// Enable axis
FB_MC2_Compact_M_nMC_Power_fbStartDelay_TON(IN:= TRUE, PT:= T#200MS, Q=> , ET=> );
IF FB_MC2_Compact_M_nMC_Power_fbStartDelay_TON.Q THEN
	IF _stAXIS_REF.NcToPlc.AxisID > 0 THEN
		IF (bE_StopDelay AND (bE_Stop OR _stAXIS_REF.Status.Moving)) THEN
			FB_MC2_Compact_M_nMC_Power_fbMC2_Power(Axis:= _stAXIS_REF, Enable:= bEnable, Enable_Positive:= bEnable_Positive, Enable_Negative:= bEnable_Negative, Override:= FB_MC2_Compact_M_nMC_Power_lrOverride, BufferMode:= MC_Aborting); 					
		ELSE
			FB_MC2_Compact_M_nMC_Power_fbMC2_Power(Axis:= _stAXIS_REF, Enable:= FALSE, Enable_Positive:= bEnable_Positive, Enable_Negative:= bEnable_Negative, Override:= FB_MC2_Compact_M_nMC_Power_lrOverride, BufferMode:= MC_Aborting); 					
		END_IF
	ELSE
		FB_MC2_Compact_M_nMC_Power_fbMC2_Power(Axis:= _stAXIS_REF, Enable:= FALSE, Enable_Positive:= bEnable_Positive, Enable_Negative:= bEnable_Negative, Override:= FB_MC2_Compact_M_nMC_Power_lrOverride, BufferMode:= MC_Aborting); 					
		IF bEnable THEN
			M_nMC_Power:= Tc3_HBI_System.cMAPPING_ERROR;
		END_IF
		RETURN;
	END_IF	 	
ELSE
	FB_MC2_Compact_M_nMC_Power_fbMC2_Power(Axis:= _stAXIS_REF, Enable:= FALSE, Enable_Positive:= bEnable_Positive, Enable_Negative:= bEnable_Negative, Override:= FB_MC2_Compact_M_nMC_Power_lrOverride, BufferMode:= MC_Aborting); 					
END_IF


// Error handling
IF FB_MC2_Compact_M_nMC_Power_fbMC2_Power.Error THEN
	M_nError(nErrorID:= FB_MC2_Compact_M_nMC_Power_fbMC2_Power.ErrorID);
	_sMessage:= 'Axis Power Error';
END_IF

// Local error
IF NOT _bError AND NOT _bReset THEN
	FB_MC2_Compact_M_nMC_Power_bError:= FALSE;
END_IF
IF _bError THEN
	FB_MC2_Compact_M_nMC_Power_bError:= TRUE;
END_IF

//**************************************
// Status
//**************************************
THIS^._bReady:= bEnable AND _stAXIS_REF.Status.ControlLoopClosed AND NOT FB_MC2_Compact_M_nMC_Power_bError AND FB_MC2_Compact_M_nMC_Power_fbMC2_Power.Status;	// Axis ready to run

//**************************************
// Local reset
//**************************************
FB_MC2_Compact_M_nMC_Power_arr_fb_R_TRIG[1](CLK:= bEnable);
FB_MC2_Compact_M_nMC_Power_arr_fb_R_TRIG[2](CLK:= NOT bEnable);
FB_MC2_Compact_M_nMC_Power_arr_fb_R_TRIG[3](CLK:= bE_Stop);
FB_MC2_Compact_M_nMC_Power_arr_fb_R_TRIG[4](CLK:= NOT bE_Stop);
FB_MC2_Compact_M_nMC_Power_arr_fb_R_TRIG[5](CLK:= bE_StopDelay);
FB_MC2_Compact_M_nMC_Power_arr_fb_R_TRIG[6](CLK:= NOT bE_StopDelay);
FB_MC2_Compact_M_nMC_Power_arr_fb_R_TRIG[7](CLK:= NOT bEnable_Positive);
FB_MC2_Compact_M_nMC_Power_arr_fb_R_TRIG[8](CLK:= NOT bEnable_Negative);
FB_MC2_Compact_M_nMC_Power_arr_fb_R_TRIG[9](CLK:= _bAuto);
FB_MC2_Compact_M_nMC_Power_arr_fb_R_TRIG[10](CLK:= NOT _bAuto);
FB_MC2_Compact_M_nMC_Power_arr_fb_R_TRIG[11](CLK:= _bManual);
FB_MC2_Compact_M_nMC_Power_arr_fb_R_TRIG[12](CLK:= NOT _bManual);

FB_MC2_Compact_M_nMC_Power_bLocal_Halt:= FALSE;
FOR _iIdx:= 1 TO 12 DO
	IF FB_MC2_Compact_M_nMC_Power_arr_fb_R_TRIG[_iIdx].Q THEN
		FB_MC2_Compact_M_nMC_Power_bLocal_Halt:= TRUE;
	END_IF
END_FOR

//************************************
// Call methods
//************************************
IF THIS^._stAXIS_REF.Status.ControlLoopClosed THEN
 	FB_MC2_Compact_M_nMC_Power_arr_nRet[1]:= M_nMC_Local_Halt(bExecute:= NOT FB_MC2_Compact_M_nMC_QuickStop_bQuickStopRunning AND FB_MC2_Compact_M_nMC_Power_bLocal_Halt);
ELSE
	M_nMC_Local_Halt(bExecute:= FALSE);
END_IF
FB_MC2_Compact_M_nMC_Power_arr_nRet[2]:= M_nMC_ReadDriveAddress(bExecute:= bEnable);


// Error handling
IF _stAXIS_REF.Status.Error THEN
	M_nError(_stAXIS_REF.Status.ErrorID);
	M_nMC_Power:= _nErrorID;
ELSE
	FOR _iIdx:= 1 TO UINT_TO_INT(SIZEOF(FB_MC2_Compact_M_nMC_Power_arr_nRet) / SIZEOF(FB_MC2_Compact_M_nMC_Power_arr_nRet[1])) DO
		IF FB_MC2_Compact_M_nMC_Power_arr_nRet[_iIdx] > 10 THEN
			M_nError(nErrorID:= FB_MC2_Compact_M_nMC_Power_arr_nRet[_iIdx]);
			EXIT;
		END_IF
	END_FOR

	// Method return value
	IF _bError THEN
		M_nMC_Power:= _nErrorID;
	ELSE
		IF FB_MC2_Compact_M_nMC_Power_fbMC2_Power.Status THEN
			M_nMC_Power:= Tc3_HBI_System.cCOMPLETE;
		ELSE
			M_nMC_Power:= Tc3_HBI_System.cIDLE;
		END_IF
	END_IF

END_IF
END_METHOD

//	The result of the method is an unsigned double integer
//	0 = idle 
//	1 = coupled
//	2 = starting
//	3 = running
//	4 = aborted
// 	5 = no hardware connected
// 	6 = Spare
//	7 = pointer or index error
//	8 = mapping error
//	9 = parameter error
//	10 = complete
//	Any other number = ErrorID
METHOD PUBLIC M_nMC_QuickStop : UDINT
VAR_INPUT
	bExecute: BOOL;
	lrDeceleration: LREAL;
	lrJerk: LREAL;
END_VAR
// Local variable
FB_MC2_Compact_M_nMC_QuickStop_bExecute:= bExecute;
FB_MC2_Compact_M_nMC_QuickStop_lrDeceleration:= lrDeceleration;
FB_MC2_Compact_M_nMC_QuickStop_lrJerk:= lrJerk;

//**********************************
// Reset 
//**********************************
IF _bReset THEN
	IF _bError THEN
		FB_MC2_Compact_M_nMC_QuickStop_fbMC2_Stop(Axis:= _stAXIS_REF, Execute:= FALSE); 
		FB_MC2_Compact_M_nMC_QuickStop_iState:= 000;
		_sMessage:= '';
	END_IF
END_IF

//**********************************
// Wait for execute
//**********************************
IF _stAXIS_REF.NcToPlc.AxisID > 0 THEN
	FB_MC2_Compact_M_nMC_QuickStop_fbExecute_R_TRIG(CLK:= FB_MC2_Compact_M_nMC_QuickStop_bExecute);
	IF FB_MC2_Compact_M_nMC_QuickStop_fbExecute_R_TRIG.Q THEN
		FB_MC2_Compact_M_nMC_QuickStop_fbMC2_Stop(Axis:= _stAXIS_REF, Execute:= FALSE, Deceleration:= FB_MC2_Compact_M_nMC_QuickStop_lrDeceleration, Jerk:= FB_MC2_Compact_M_nMC_QuickStop_lrJerk); 
		FB_MC2_Compact_M_nMC_QuickStop_bQuickStopRunning:= TRUE;
		
		// Axis not coupled	
		IF NOT _stAXIS_REF.Status.Coupled THEN
			IF _stAXIS_REF.Status.ControlLoopClosed THEN
				IF _stAXIS_REF.Status.HasJob THEN
					FB_MC2_Compact_M_nMC_QuickStop_fbMC2_Stop.Execute:= TRUE;
					FB_MC2_Compact_M_nMC_QuickStop_iState:= 001;
				ELSE
					FB_MC2_Compact_M_nMC_QuickStop_iState:= 020;
				END_IF
			ELSE
				FB_MC2_Compact_M_nMC_QuickStop_iState:= 020;
			END_IF
		ELSE
			FB_MC2_Compact_M_nMC_QuickStop_iState:= 010;
		END_IF
	END_IF
ELSE
	FB_MC2_Compact_M_nMC_QuickStop_fbExecute_R_TRIG(CLK:= FALSE);
	FB_MC2_Compact_M_nMC_QuickStop_iState:= 000;
	IF FB_MC2_Compact_M_nMC_QuickStop_bExecute THEN
		M_nMC_QuickStop:= Tc3_HBI_System.cMAPPING_ERROR;
	END_IF
	RETURN;
END_IF


//**********************************
// Main sequence
//**********************************
CASE FB_MC2_Compact_M_nMC_QuickStop_iState OF

	000: 	// Do nothing
			FB_MC2_Compact_M_nMC_QuickStop_bQuickStopRunning:= FALSE;
	
	001:	// Stop Axis
			M_nMC_QuickStop:= Tc3_HBI_System.cRUNNING;
			FB_MC2_Compact_M_nMC_QuickStop_fbMC2_Stop(Axis:= _stAXIS_REF); 
			
			// Stop Axis
			IF _stAXIS_REF.Status.PTPmode AND _stAXIS_REF.Status.Operational THEN
				FB_MC2_Compact_M_nMC_QuickStop_fbMC2_Stop.Execute:= TRUE; 
		
				// Command aborted
				IF FB_MC2_Compact_M_nMC_QuickStop_fbMC2_Stop.CommandAborted THEN
					FB_MC2_Compact_M_nMC_QuickStop_iState:= 020;
				ELSE
					// Error handling
					IF FB_MC2_Compact_M_nMC_QuickStop_fbMC2_Stop.Error THEN
						M_nError(nErrorID:= FB_MC2_Compact_M_nMC_QuickStop_fbMC2_Stop.ErrorID);
						M_nMC_QuickStop:= FB_MC2_Compact_M_nMC_QuickStop_fbMC2_Stop.ErrorID;
						_sMessage:= 'Axis Quick Stop Error';
					ELSE
						// Done
						IF FB_MC2_Compact_M_nMC_QuickStop_fbMC2_Stop.Done THEN
							FB_MC2_Compact_M_nMC_QuickStop_fbMC2_Stop(Axis:= _stAXIS_REF, Execute:= FALSE); 
							FB_MC2_Compact_M_nMC_QuickStop_iState:= 020;
						END_IF
					END_IF
				END_IF
			ELSE
				FB_MC2_Compact_M_nMC_QuickStop_iState:= 020;
			END_IF
	
	010:	// Coupled
			M_nMC_QuickStop:= Tc3_HBI_System.cCOUPLED;
			FB_MC2_Compact_M_nMC_QuickStop_fbMC2_Stop(Axis:= _stAXIS_REF); 
			FB_MC2_Compact_M_nMC_QuickStop_bQuickStopRunning:= FALSE;

			IF NOT FB_MC2_Compact_M_nMC_QuickStop_bExecute THEN
				FB_MC2_Compact_M_nMC_QuickStop_fbMC2_Stop(Axis:= _stAXIS_REF, Execute:= FALSE); 
				FB_MC2_Compact_M_nMC_QuickStop_iState:= 000;
			END_IF	

	020:	// Done
			M_nMC_QuickStop:= Tc3_HBI_System.cCOMPLETE;
			FB_MC2_Compact_M_nMC_QuickStop_fbMC2_Stop(Axis:= _stAXIS_REF); 
			FB_MC2_Compact_M_nMC_QuickStop_bQuickStopRunning:= FALSE;

			IF FB_MC2_Compact_M_nMC_QuickStop_bExecute THEN
				IF FB_MC2_Compact_M_nMC_QuickStop_fbMC2_Stop.CommandAborted THEN
					M_nMC_QuickStop:= Tc3_HBI_System.cABORTED;
				END_IF
			ELSE
				FB_MC2_Compact_M_nMC_QuickStop_fbMC2_Stop(Axis:= _stAXIS_REF, Execute:= FALSE); 
				FB_MC2_Compact_M_nMC_QuickStop_iState:= 000;
			END_IF	
		
ELSE
	FB_MC2_Compact_M_nMC_QuickStop_iState:= 000;
END_CASE
END_METHOD

//	The result of the method is an unsigned double integer
//	0 = idle 
//	1 = coupled
//	2 = starting
//	3 = running
//	4 = aborted
// 	5 = no hardware connected
// 	6 = Spare
//	7 = pointer or index error
//	8 = mapping error
//	9 = parameter error
//	10 = complete
//	Any other number = ErrorID
METHOD PRIVATE M_nMC_ReadDriveAddress : UDINT
VAR_INPUT
	bExecute: BOOL;
END_VAR
// Local variable
FB_MC2_Compact_M_nMC_ReadDriveAddress_bExecute:= bExecute;

//**********************************
// Reset 
//**********************************
IF _bReset THEN
	FB_MC2_Compact_M_nMC_ReadDriveAddress_iState:= 000;
	_sMessage:= '';
END_IF

// Check for Axis
IF _stAXIS_REF.NcToPlc.AxisID = 0 THEN
	Tc2_System.MEMSET(destAddr:= ADR(_stDriveAddress), fillByte:= 16#00, n:= SIZEOF(_stDriveAddress));	
	FB_MC2_Compact_M_nMC_ReadDriveAddress_iState:= 000;
	IF FB_MC2_Compact_M_nMC_ReadDriveAddress_bExecute THEN
		M_nMC_ReadDriveAddress:= Tc3_HBI_System.cMAPPING_ERROR;
	END_IF
	RETURN;
END_IF

//**********************************
// Main sequence
//**********************************
CASE FB_MC2_Compact_M_nMC_ReadDriveAddress_iState OF

	000: 	// Init
			M_nMC_ReadDriveAddress:= Tc3_HBI_System.cSTARTING;
			FB_MC2_Compact_M_nMC_ReadDriveAddress_fbReadDriveAddress(Axis:= _stAXIS_REF, Execute:= FALSE);
			
			// WcState ok 
			IF NOT BIT_TO_BOOL(_stAXIS_REF.NcToPlc.StateDWord.30) AND NOT _stAXIS_REF.Status.OpMode.SimulationAxis THEN
				// Axis connected to Hardware
				IF _stAXIS_REF.NcToPlc.AxisID > 0 THEN
					FB_MC2_Compact_M_nMC_ReadDriveAddress_iState:= FB_MC2_Compact_M_nMC_ReadDriveAddress_iState +1;
				END_IF	
			END_IF	
		
	001:	// Read drive address		
			M_nMC_ReadDriveAddress:= Tc3_HBI_System.cSTARTING;
			FB_MC2_Compact_M_nMC_ReadDriveAddress_fbReadDriveAddress(Axis:= _stAXIS_REF, Execute:= TRUE);
			FB_MC2_Compact_M_nMC_ReadDriveAddress_iState:= FB_MC2_Compact_M_nMC_ReadDriveAddress_iState +1;

	002:	// Read drive address done	
			M_nMC_ReadDriveAddress:= Tc3_HBI_System.cRUNNING;
			FB_MC2_Compact_M_nMC_ReadDriveAddress_fbReadDriveAddress(Axis:= _stAXIS_REF, Execute:= TRUE);
			
			// Error
			IF FB_MC2_Compact_M_nMC_ReadDriveAddress_fbReadDriveAddress.Error THEN
				M_nError(nErrorID:= FB_MC2_Compact_M_nMC_ReadDriveAddress_fbReadDriveAddress.ErrorID);
				M_nMC_ReadDriveAddress:= FB_MC2_Compact_M_nMC_ReadDriveAddress_fbReadDriveAddress.ErrorID;
				_sMessage:= 'Axis Read Drive Address Error';
			ELSE
				// Done
				IF NOT FB_MC2_Compact_M_nMC_ReadDriveAddress_fbReadDriveAddress.Busy AND FB_MC2_Compact_M_nMC_ReadDriveAddress_fbReadDriveAddress.Done THEN
					_stDriveAddress:= FB_MC2_Compact_M_nMC_ReadDriveAddress_fbReadDriveAddress.DriveAddress;
					FB_MC2_Compact_M_nMC_ReadDriveAddress_fbReadDriveAddress(Axis:= _stAXIS_REF, Execute:= FALSE);
					FB_MC2_Compact_M_nMC_ReadDriveAddress_iState:= FB_MC2_Compact_M_nMC_ReadDriveAddress_iState +1;
				END_IF
			END_IF
	
	003: // Done
			M_nMC_ReadDriveAddress:= Tc3_HBI_System.cCOMPLETE;

ELSE
	FB_MC2_Compact_M_nMC_ReadDriveAddress_iState:= 000;
END_CASE
END_METHOD

//	The result of the method is an unsigned double integer
//	0 = idle 
//	1 = coupled
//	2 = starting
//	3 = running
//	4 = aborted
// 	5 = no hardware connected
// 	6 = Spare
//	7 = pointer or index error
//	8 = mapping error
//	9 = parameter error
//	10 = complete
//	Any other number = ErrorID
METHOD PUBLIC M_nMC_Stop : UDINT
VAR_INPUT
	bExecute: BOOL;
END_VAR
// Local variable
FB_MC2_Compact_M_nMC_Stop_bExecute:= bExecute;

//**********************************
// Reset 
//**********************************
IF _bReset THEN
	IF _bError THEN
		FB_MC2_Compact_M_nMC_Stop_fbMC2_Stop1(Axis:= _stAXIS_REF, Execute:= FALSE);
		FB_MC2_Compact_M_nMC_Stop_fbMC2_Stop2(Axis:= _stAXIS_REF, Execute:= FALSE);
		FB_MC2_Compact_M_nMC_Stop_iState:= 000;
		_sMessage:= '';
	END_IF
END_IF

//**********************************
// Wait for execute
//**********************************
IF _stAXIS_REF.NcToPlc.AxisID > 0 THEN
	FB_MC2_Compact_M_nMC_Stop_fbExecute_R_TRIG(CLK:= FB_MC2_Compact_M_nMC_Stop_bExecute);
	IF FB_MC2_Compact_M_nMC_Stop_fbExecute_R_TRIG.Q THEN
		FB_MC2_Compact_M_nMC_Stop_fbMC2_Stop1(Axis:= _stAXIS_REF, Deceleration:= _stDynamic.lrDeceleration, Jerk:= _stDynamic.lrJerk); 
		FB_MC2_Compact_M_nMC_Stop_fbMC2_Stop2(Axis:= _stAXIS_REF, Deceleration:= _stDynamic.lrDeceleration, Jerk:= _stDynamic.lrJerk); 
		
		// Axis not coupled	
		IF NOT _stAXIS_REF.Status.Coupled THEN
			IF FB_MC2_Compact_M_nMC_Stop_fbMC2_Stop1.Execute OR FB_MC2_Compact_M_nMC_Stop_fbMC2_Stop1.Busy THEN
				FB_MC2_Compact_M_nMC_Stop_fbMC2_Stop1(Axis:= _stAXIS_REF, Execute:= FALSE); 
				FB_MC2_Compact_M_nMC_Stop_fbMC2_Stop2(Axis:= _stAXIS_REF, Execute:= FALSE); 
				FB_MC2_Compact_M_nMC_Stop_fbMC2_Stop2.Execute:= TRUE;
				FB_MC2_Compact_M_nMC_Stop_iState:= 010;
			ELSE
				FB_MC2_Compact_M_nMC_Stop_fbMC2_Stop1(Axis:= _stAXIS_REF, Execute:= FALSE); 
				FB_MC2_Compact_M_nMC_Stop_fbMC2_Stop2(Axis:= _stAXIS_REF, Execute:= FALSE); 
				FB_MC2_Compact_M_nMC_Stop_fbMC2_Stop1.Execute:= TRUE;
				FB_MC2_Compact_M_nMC_Stop_iState:= 001;
			END_IF
		ELSE
			FB_MC2_Compact_M_nMC_Stop_fbMC2_Stop1(Axis:= _stAXIS_REF, Execute:= FALSE); 
			FB_MC2_Compact_M_nMC_Stop_fbMC2_Stop2(Axis:= _stAXIS_REF, Execute:= FALSE); 
			FB_MC2_Compact_M_nMC_Stop_iState:= 030;
		END_IF
	
	END_IF
ELSE
	FB_MC2_Compact_M_nMC_Stop_fbExecute_R_TRIG(CLK:= FALSE);
	FB_MC2_Compact_M_nMC_Stop_iState:= 000;
	IF FB_MC2_Compact_M_nMC_Stop_bExecute THEN
		M_nMC_Stop:= Tc3_HBI_System.cMAPPING_ERROR;
	END_IF
	RETURN;
END_IF


//**********************************
// Main sequence
//**********************************
CASE FB_MC2_Compact_M_nMC_Stop_iState OF

	000: 	// Do nothing
	
	001:	// Stop Axis1
			M_nMC_Stop:= Tc3_HBI_System.cSTARTING;
			FB_MC2_Compact_M_nMC_Stop_fbMC2_Stop1(Axis:= _stAXIS_REF);
			FB_MC2_Compact_M_nMC_Stop_fbMC2_Stop2(Axis:= _stAXIS_REF);
	
			// Command aborted
			IF FB_MC2_Compact_M_nMC_Stop_fbMC2_Stop1.CommandAborted THEN
				FB_MC2_Compact_M_nMC_Stop_fbMC2_Stop2.Execute:= FALSE;
				FB_MC2_Compact_M_nMC_Stop_iState:= 040;
			ELSE
				// Error handling
				IF FB_MC2_Compact_M_nMC_Stop_fbMC2_Stop1.Error THEN
					M_nError(FB_MC2_Compact_M_nMC_Stop_fbMC2_Stop1.ErrorID);
					M_nMC_Stop:= FB_MC2_Compact_M_nMC_Stop_fbMC2_Stop1.ErrorID;
					_sMessage:= 'Axis Stop Error';
				ELSE
					// Active
					IF FB_MC2_Compact_M_nMC_Stop_fbMC2_Stop1.Active THEN
						FB_MC2_Compact_M_nMC_Stop_iState:= 02;
					ELSE
						// Done
						IF FB_MC2_Compact_M_nMC_Stop_fbMC2_Stop1.Done THEN
							FB_MC2_Compact_M_nMC_Stop_iState:= 040;
						END_IF
					END_IF	
				END_IF
			END_IF

	002:	// Stop Axis
			M_nMC_Stop:= Tc3_HBI_System.cRUNNING;
			FB_MC2_Compact_M_nMC_Stop_fbMC2_Stop1(Axis:= _stAXIS_REF);
			FB_MC2_Compact_M_nMC_Stop_fbMC2_Stop2(Axis:= _stAXIS_REF);
	
			// Command aborted
			IF FB_MC2_Compact_M_nMC_Stop_fbMC2_Stop1.CommandAborted THEN
				FB_MC2_Compact_M_nMC_Stop_fbMC2_Stop2.Execute:= FALSE;
				FB_MC2_Compact_M_nMC_Stop_iState:= 040;
			ELSE
				// Error handling
				IF FB_MC2_Compact_M_nMC_Stop_fbMC2_Stop1.Error THEN
					M_nError(FB_MC2_Compact_M_nMC_Stop_fbMC2_Stop1.ErrorID);
					M_nMC_Stop:= FB_MC2_Compact_M_nMC_Stop_fbMC2_Stop1.ErrorID;
					_sMessage:= 'Axis Stop Error';
				ELSE
					// Done
					IF FB_MC2_Compact_M_nMC_Stop_fbMC2_Stop1.Done THEN
						FB_MC2_Compact_M_nMC_Stop_iState:= 040;
					END_IF
				END_IF
			END_IF 

	010:	// Stop Axis1
			M_nMC_Stop:= Tc3_HBI_System.cSTARTING;
			FB_MC2_Compact_M_nMC_Stop_fbMC2_Stop1(Axis:= _stAXIS_REF);
			FB_MC2_Compact_M_nMC_Stop_fbMC2_Stop2(Axis:= _stAXIS_REF);
			
			// Command aborted
			IF FB_MC2_Compact_M_nMC_Stop_fbMC2_Stop2.CommandAborted THEN
				FB_MC2_Compact_M_nMC_Stop_fbMC2_Stop1.Execute:= FALSE;
				FB_MC2_Compact_M_nMC_Stop_iState:= 040;
			ELSE
				// Error handling
				IF FB_MC2_Compact_M_nMC_Stop_fbMC2_Stop2.Error THEN
					M_nError(FB_MC2_Compact_M_nMC_Stop_fbMC2_Stop2.ErrorID);
					M_nMC_Stop:= FB_MC2_Compact_M_nMC_Stop_fbMC2_Stop2.ErrorID;
					_sMessage:= 'Axis Stop Error';
				ELSE
					// Active
					IF FB_MC2_Compact_M_nMC_Stop_fbMC2_Stop2.Active THEN
						FB_MC2_Compact_M_nMC_Stop_iState:= 011;
					ELSE
						// Done
						IF FB_MC2_Compact_M_nMC_Stop_fbMC2_Stop2.Done THEN
							FB_MC2_Compact_M_nMC_Stop_iState:= 040;
						END_IF
					END_IF	
				END_IF
			END_IF 
			
	011:	// Stop Axis2
			M_nMC_Stop:= Tc3_HBI_System.cRUNNING;
			FB_MC2_Compact_M_nMC_Stop_fbMC2_Stop1(Axis:= _stAXIS_REF);
			FB_MC2_Compact_M_nMC_Stop_fbMC2_Stop2(Axis:= _stAXIS_REF);
			
			// Command aborted
			IF FB_MC2_Compact_M_nMC_Stop_fbMC2_Stop2.CommandAborted THEN
				FB_MC2_Compact_M_nMC_Stop_fbMC2_Stop1.Execute:= FALSE;
				FB_MC2_Compact_M_nMC_Stop_iState:= 040;
			ELSE
				// Error handling
				IF FB_MC2_Compact_M_nMC_Stop_fbMC2_Stop2.Error THEN
					M_nError(FB_MC2_Compact_M_nMC_Stop_fbMC2_Stop2.ErrorID);
					M_nMC_Stop:= FB_MC2_Compact_M_nMC_Stop_fbMC2_Stop2.ErrorID;
					_sMessage:= 'Axis Stop Error';
				ELSE
					// Done
					IF FB_MC2_Compact_M_nMC_Stop_fbMC2_Stop2.Done THEN
						FB_MC2_Compact_M_nMC_Stop_iState:= 040;
					END_IF
				END_IF
			END_IF
		
	030:	// Coupled
			M_nMC_Stop:= Tc3_HBI_System.cCOUPLED;
			FB_MC2_Compact_M_nMC_Stop_fbMC2_Stop1(Axis:= _stAXIS_REF);
			FB_MC2_Compact_M_nMC_Stop_fbMC2_Stop2(Axis:= _stAXIS_REF);

			IF NOT FB_MC2_Compact_M_nMC_Stop_bExecute THEN
				FB_MC2_Compact_M_nMC_Stop_fbMC2_Stop1(Axis:= _stAXIS_REF, Execute:= FALSE);
				FB_MC2_Compact_M_nMC_Stop_fbMC2_Stop2(Axis:= _stAXIS_REF, Execute:= FALSE);
				FB_MC2_Compact_M_nMC_Stop_iState:= 000;
			END_IF	

	040:	// Done
			M_nMC_Stop:= Tc3_HBI_System.cCOMPLETE;
			FB_MC2_Compact_M_nMC_Stop_fbMC2_Stop1(Axis:= _stAXIS_REF);
			FB_MC2_Compact_M_nMC_Stop_fbMC2_Stop2(Axis:= _stAXIS_REF);

			IF FB_MC2_Compact_M_nMC_Stop_bExecute THEN
				IF FB_MC2_Compact_M_nMC_Stop_fbMC2_Stop1.Execute AND FB_MC2_Compact_M_nMC_Stop_fbMC2_Stop1.CommandAborted THEN
					M_nMC_Stop:= Tc3_HBI_System.cABORTED;
				END_IF
				IF FB_MC2_Compact_M_nMC_Stop_fbMC2_Stop2.Execute AND FB_MC2_Compact_M_nMC_Stop_fbMC2_Stop2.CommandAborted THEN
					M_nMC_Stop:= Tc3_HBI_System.cABORTED;
				END_IF
			ELSE	
				FB_MC2_Compact_M_nMC_Stop_fbMC2_Stop1(Axis:= _stAXIS_REF, Execute:= FALSE);
				FB_MC2_Compact_M_nMC_Stop_fbMC2_Stop2(Axis:= _stAXIS_REF, Execute:= FALSE);
				FB_MC2_Compact_M_nMC_Stop_iState:= 000;
			END_IF	
		
ELSE
	FB_MC2_Compact_M_nMC_Stop_iState:= 000;
END_CASE
END_METHOD

//	The result of the method is an unsigned double integer
//	0 = idle 
//	1 = coupled
//	2 = starting
//	3 = running
//	4 = aborted
// 	5 = no hardware connected
// 	6 = Spare
//	7 = pointer or index error
//	8 = mapping error
//	9 = parameter error
//	10 = complete
//	Any other number = ErrorID
METHOD PUBLIC M_nReset : UDINT
VAR_INPUT
	bExecute: BOOL;
END_VAR
// Local variable
FB_MC2_Compact_M_nReset_bExecute:= bExecute;

//**********************************
// Wait for execute
//**********************************
FB_MC2_Compact_M_nReset_fbExecute_R_TRIG(CLK:= FB_MC2_Compact_M_nReset_bExecute);
IF FB_MC2_Compact_M_nReset_fbExecute_R_TRIG.Q THEN
	FB_MC2_Compact_M_nReset_fbMC2_Reset(Axis:= _stAXIS_REF, Execute:= FALSE);
	SUPER^.M_nReset(bExecute:= FALSE);
	FB_MC2_Compact_M_nReset_iState:= 001;
	_sMessage:= '';
END_IF	


//**********************************
// Main sequence
//**********************************
CASE FB_MC2_Compact_M_nReset_iState OF

	000: 	// Do nothing
		
	001:	// Reset NC
			M_nReset:= Tc3_HBI_System.cSTARTING;
			FB_MC2_Compact_M_nReset_fbMC2_Reset(Axis:= _stAXIS_REF, Execute:= FALSE);
			
			// Check for not encoder axis
			IF _stAXIS_REF.Status.ErrorID = _stAXIS_REF.NcToPlc.ErrorCode THEN
				IF _stAXIS_REF.Status.Error THEN
					IF _stAXIS_REF.Status.Coupled THEN
						FB_MC2_Compact_M_nReset_iState:= FB_MC2_Compact_M_nReset_iState +2;
					ELSE
						IF _stAXIS_REF.Status.Error OR NOT _stAXIS_REF.Status.HasJob THEN 
							FB_MC2_Compact_M_nReset_iState:= FB_MC2_Compact_M_nReset_iState +1;
						ELSE
							FB_MC2_Compact_M_nReset_iState:= FB_MC2_Compact_M_nReset_iState +2;
						END_IF	
					END_IF
				ELSE
					FB_MC2_Compact_M_nReset_iState:= FB_MC2_Compact_M_nReset_iState +2;
				END_IF
			ELSE
				// Encoder axis
				FB_MC2_Compact_M_nReset_iState:= FB_MC2_Compact_M_nReset_iState +1;
			END_IF
	
	002:	// Reset NC
			M_nReset:= Tc3_HBI_System.cRUNNING;
			FB_MC2_Compact_M_nReset_fbMC2_Reset(Axis:= _stAXIS_REF, Execute:= TRUE); 
	
			// Error handling
			IF FB_MC2_Compact_M_nReset_fbMC2_Reset.Error THEN
				M_nError(FB_MC2_Compact_M_nReset_fbMC2_Reset.ErrorID);
				M_nReset:= FB_MC2_Compact_M_nReset_fbMC2_Reset.ErrorID;
				FB_MC2_Compact_M_nReset_iState:= FB_MC2_Compact_M_nReset_iState +1;
				_sMessage:= 'Axis Reset Error';
			ELSE
				// Done
				IF FB_MC2_Compact_M_nReset_fbMC2_Reset.Done THEN
					FB_MC2_Compact_M_nReset_iState:= FB_MC2_Compact_M_nReset_iState +1;
				END_IF
			END_IF
		
	003:	// Reset father	
			M_nReset:= Tc3_HBI_System.cRUNNING;
			FB_MC2_Compact_M_nReset_nStatus:= SUPER^.M_nReset(bExecute:= TRUE);
			
			// Error handling
			IF FB_MC2_Compact_M_nReset_nStatus > Tc3_HBI_System.cCOMPLETE THEN
				SUPER^.M_nReset(bExecute:= FALSE);		
				IF _stAXIS_REF.Status.Coupled THEN
					FB_MC2_Compact_M_nReset_iState:= 020;
				ELSE
					FB_MC2_Compact_M_nReset_iState:= 030;
				END_IF
			END_IF

			// Done
			IF FB_MC2_Compact_M_nReset_nStatus = Tc3_HBI_System.cCOUPLED OR FB_MC2_Compact_M_nReset_nStatus = Tc3_HBI_System.cCOMPLETE THEN
				SUPER^.M_nReset(bExecute:= FALSE);		
				IF _stAXIS_REF.Status.Coupled THEN
					FB_MC2_Compact_M_nReset_iState:= 020;
				ELSE
					FB_MC2_Compact_M_nReset_iState:= 030;
				END_IF
			END_IF
			
	020:	// Coupled
			M_nReset:= Tc3_HBI_System.cCOUPLED;
			IF NOT FB_MC2_Compact_M_nReset_bExecute THEN
				FB_MC2_Compact_M_nReset_fbMC2_Reset(Axis:= _stAXIS_REF, Execute:= FALSE);
				SUPER^.M_nReset(bExecute:= FALSE);		
				FB_MC2_Compact_M_nReset_iState:= 000;
			END_IF	
	
	030:	// Done
			M_nReset:= Tc3_HBI_System.cCOMPLETE;
			IF NOT FB_MC2_Compact_M_nReset_bExecute THEN
				FB_MC2_Compact_M_nReset_fbMC2_Reset(Axis:= _stAXIS_REF, Execute:= FALSE);
				SUPER^.M_nReset(bExecute:= FALSE);		
				FB_MC2_Compact_M_nReset_iState:= 000;
			END_IF

ELSE
	FB_MC2_Compact_M_nReset_iState:= 000;
END_CASE
END_METHOD

PROPERTY PUBLIC P_bE_Stop : BOOL
GET
P_bE_Stop:= FB_MC2_Compact_M_nMC_Power_bE_Stop;
END_GET
END_PROPERTY

PROPERTY PUBLIC P_bE_StopDelay : BOOL
GET
P_bE_StopDelay:= FB_MC2_Compact_M_nMC_Power_bE_StopDelay;
END_GET
END_PROPERTY

PROPERTY PUBLIC P_bEnable : BOOL
GET
P_bEnable:= FB_MC2_Compact_M_nMC_Power_bEnable;
END_GET
END_PROPERTY

PROPERTY PUBLIC P_bEnable_Negative : BOOL
GET
P_bEnable_Negative:= FB_MC2_Compact_M_nMC_Power_bEnable_Negative;
END_GET
END_PROPERTY

PROPERTY PUBLIC P_bEnable_Positive : BOOL
GET
P_bEnable_Positive:= FB_MC2_Compact_M_nMC_Power_bEnable_Positive;
END_GET
END_PROPERTY

PROPERTY PUBLIC P_bHardwareConnected : BOOL
GET
P_bHardwareConnected:= _bHardwareConnected;
END_GET
END_PROPERTY

PROPERTY PUBLIC P_bHomed : BOOL
GET
P_bHomed:= _stAXIS_REF.Status.Homed;
END_GET
END_PROPERTY

PROPERTY PUBLIC P_eBufferMode : MC_BufferMode
SET
_eBufferMode:= P_eBufferMode;
END_SET
END_PROPERTY

PROPERTY PUBLIC P_lrOverride : LREAL
GET
PUBLIC 
VAR
END_VAR
P_lrOverride:= FB_MC2_Compact_M_nMC_Power_lrOverride;
END_GET
SET
IF P_lrOverride < 0.0 THEN
	FB_MC2_Compact_M_nMC_Power_lrOverride:= 0.0;
ELSE
	IF 	P_lrOverride > 100.0 THEN
		FB_MC2_Compact_M_nMC_Power_lrOverride:= 100.0;
	ELSE
		FB_MC2_Compact_M_nMC_Power_lrOverride:= P_lrOverride;
	END_IF
END_IF
END_SET
END_PROPERTY

PROPERTY PUBLIC P_pAXIS_REF : POINTER TO AXIS_REF
GET
P_pAXIS_REF:= ADR(_stAXIS_REF);
END_GET
END_PROPERTY

PROPERTY PUBLIC P_pDriveAddress : POINTER TO ST_AdsAddress
GET
P_pDriveAddress:= ADR(_stDriveAddress);
END_GET
END_PROPERTY

PROPERTY PUBLIC P_sMessage : STRING
GET
P_sMessage:= _sMessage;
END_GET
END_PROPERTY

PROPERTY PUBLIC P_stDynamic : _ST_MC2_Dynamic
GET
P_stDynamic:= _stDynamic;
END_GET
END_PROPERTY

END_FUNCTION_BLOCK

// MOTION/POUs/FBs/Basic/FB_MC2_AX8000
//------------------------------------------------------------------------------------------
//                                                                                        	
//***************************** Beckhoff TwinCAT Examples **********************************
//                                                                                        	
//************************************* WARNING ********************************************
// This program is only an example. If it is used as a control program in any real        	
// application, Beckhoff is not responsible for any malfunction, loss or damage           	
// which could arise by using this program!                                               	
//                                                                                        	
//*************************************  Program Info. *************************************
//                                                                                        	
// PLC program name:    	FB_MC2_Basic_AX8000 (FB)               	                           	
// Hardware platform:      	TwinCat PTP v3.1 4022				                          	                                  	
//                                                                                        	
// ======================================================================================== 
//         Version       Date                        Remarks                              	
// ======================================================================================== 
//         3.1           27 feb 2018                 First release of this example        	
//
// ======================================================================================== 
//                                                                                        	
//******************************* Aims OF this PLC PROGRAM *********************************
//                                                                                        	
// MC2 AX8000 servo axis 						 			                               	
//                                                                                        	
//----------------------------------------------------------------------------------------- 
FUNCTION_BLOCK FB_MC2_AX8000 EXTENDS FB_MC2_Basic 
VAR
	FB_MC2_AX8000_M_nMC_Brake_bExecute: BOOL;
	FB_MC2_AX8000_M_nMC_Brake_eBrakeState: E_MC2_AX8000_Brake;
	FB_MC2_AX8000_M_nMC_Brake_iState: INT;
	FB_MC2_AX8000_M_nMC_Brake_nValue: UINT;
	FB_MC2_AX8000_M_nMC_Brake_fbExecute_R_TRIG: Tc2_Standard.R_TRIG;
	FB_MC2_AX8000_M_nMC_Brake_fbCoEWrite: Tc2_MC2_Drive.FB_CoEWrite;

	FB_MC2_AX8000_M_nMC_DriveData_iState: INT;	
	FB_MC2_AX8000_M_nMC_DriveData_lrActualMainVoltage: LREAL;
	FB_MC2_AX8000_M_nMC_DriveData_lrAmplifierTemperature: LREAL;
	FB_MC2_AX8000_M_nMC_DriveData_lrMotorTemperature: LREAL;
	FB_MC2_AX8000_M_nMC_DriveData_fbCoERead: Tc2_MC2_Drive.FB_CoERead;
	FB_MC2_AX8000_M_nMC_DriveData_fbCoEWrite: Tc2_MC2_Drive.FB_CoEWrite;
	FB_MC2_AX8000_M_nMC_DriveData_iValue: INT;
	FB_MC2_AX8000_M_nMC_DriveData_rValue: REAL;
	
	FB_MC2_AX8000_M_nMC_Power_bEnable: BOOL;
	FB_MC2_AX8000_M_nMC_Power_bE_Stop: BOOL;
	FB_MC2_AX8000_M_nMC_Power_bE_StopDelay: BOOL;
	FB_MC2_AX8000_M_nMC_Power_bEnable_Positive: BOOL;
	FB_MC2_AX8000_M_nMC_Power_bEnable_Negative: BOOL;
	FB_MC2_AX8000_M_nMC_Power_fbStartDelay_TON: Tc2_Standard.TON;
	FB_MC2_AX8000_M_nMC_Power_arr_nRet: ARRAY[1..4] OF UDINT;

	FB_MC2_AX8000_M_nMC_Torque_bExecute: BOOL;
	FB_MC2_AX8000_M_nMC_Torque_lrTorque: LREAL; 		// Torque limit 0.0-500.0%	
	FB_MC2_AX8000_M_nMC_Torque_iState: INT;
	FB_MC2_AX8000_M_nMC_Torque_iTorque: INT;
	FB_MC2_AX8000_M_nMC_Torque_fbExecute_R_TRIG: R_TRIG;
	FB_MC2_AX8000_M_nMC_Torque_fbCoEWrite: Tc2_MC2_Drive.FB_CoEWrite;
	
	FB_MC2_AX8000_M_nReset_iState: INT;
	FB_MC2_AX8000_M_nReset_fbExecute_R_TRIG: Tc2_Standard.R_TRIG;
	FB_MC2_AX8000_M_nReset_nStatus: UDINT;
END_VAR

//	The result of the method is an unsigned double integer
//	0 = idle 
//	1 = coupled
//	2 = starting
//	3 = running
//	4 = aborted
// 	5 = no hardware connected
// 	6 = Spare
//	7 = pointer or index error
//	8 = mapping error
//	9 = parameter error
//	10 = complete
//	Any other number = ErrorID
METHOD PUBLIC M_nMC_Brake : UDINT
VAR_INPUT
	bExecute: BOOL;
	eBrakeState: E_MC2_AX8000_Brake;
END_VAR
// Local variable
FB_MC2_AX8000_M_nMC_Brake_bExecute:= bExecute;
FB_MC2_AX8000_M_nMC_Brake_eBrakeState:= eBrakeState;

//**********************************
// Reset 
//**********************************
IF _bReset THEN
	IF _bError THEN
		FB_MC2_AX8000_M_nMC_Brake_fbCoEWrite(Execute:= FALSE, Axis:= _stAXIS_REF); 
		FB_MC2_AX8000_M_nMC_Brake_iState:= 000;
	END_IF
END_IF

// No hardware connected
IF NOT _bHardwareConnected THEN
	FB_MC2_AX8000_M_nMC_Brake_fbCoEWrite(Execute:= FALSE, Axis:= _stAXIS_REF); 
	FB_MC2_AX8000_M_nMC_Brake_iState:= 000;
	IF FB_MC2_AX8000_M_nMC_Brake_bExecute THEN
		M_nMC_Brake:= Tc3_HBI_System.cNO_HARDWARE_CONNECTED;
	END_IF	
	RETURN;
END_IF

// Parameter check 
IF FB_MC2_AX8000_M_nMC_Brake_bExecute THEN
	IF FB_MC2_AX8000_M_nMC_Brake_eBrakeState = AX8000_Brake_Release_force OR FB_MC2_AX8000_M_nMC_Brake_eBrakeState = AX8000_Brake_Force_lock OR FB_MC2_AX8000_M_nMC_Brake_eBrakeState = AX8000_Brake_Force_unlock THEN
		;
	ELSE
		// Parameter error	
		M_nMC_Brake:= Tc3_HBI_System.cPARAMETER_ERROR;
		RETURN;
	END_IF
END_IF

//**********************************
// Wait for execute
//**********************************
IF _stAXIS_REF.NcToPlc.AxisID > 0 THEN
	FB_MC2_AX8000_M_nMC_Brake_fbExecute_R_TRIG(CLK:= FB_MC2_AX8000_M_nMC_Brake_bExecute);
	IF FB_MC2_AX8000_M_nMC_Brake_fbExecute_R_TRIG.Q THEN
		FB_MC2_AX8000_M_nMC_Brake_fbCoEWrite(Execute:= FALSE, Axis:= _stAXIS_REF); 
		FB_MC2_AX8000_M_nMC_Brake_iState:= 001;
	END_IF
ELSE
	FB_MC2_AX8000_M_nMC_Brake_iState:= 000;
	IF FB_MC2_AX8000_M_nMC_Brake_bExecute THEN
		M_nMC_Brake:= Tc3_HBI_System.cMAPPING_ERROR;		
	END_IF
	RETURN;
END_IF


//**********************************
// Main sequence
//**********************************
CASE FB_MC2_AX8000_M_nMC_Brake_iState OF

	000: 	// Do nothing
	
	001:	// Set brake state
			M_nMC_Brake:= Tc3_HBI_System.cRUNNING;

			CASE FB_MC2_AX8000_M_nMC_Brake_eBrakeState OF
				
				AX8000_Brake_Release_force:
					FB_MC2_AX8000_M_nMC_Brake_nValue:= 0;

				AX8000_Brake_Force_lock:
					FB_MC2_AX8000_M_nMC_Brake_nValue:= 1;
			
				AX8000_Brake_Force_unlock:
					FB_MC2_AX8000_M_nMC_Brake_nValue:= 2;
				
			ELSE	
				FB_MC2_AX8000_M_nMC_Brake_nValue:= 0;
			END_CASE

			FB_MC2_AX8000_M_nMC_Brake_iState:= FB_MC2_AX8000_M_nMC_Brake_iState +1;

	002:	// Write brake state to AX8000
			M_nMC_Brake:= Tc3_HBI_System.cRUNNING;
			FB_MC2_AX8000_M_nMC_Brake_fbCoEWrite(Execute:= FALSE, Axis:= _stAXIS_REF); 
			FB_MC2_AX8000_M_nMC_Brake_fbCoEWrite(
				NetId:= '', 
				Index:= 16#3000 + (16#0400 * _stDriveAddress.Channel), 
				SubIndex:= 16#07, 
				pSrcBuf:= ADR(FB_MC2_AX8000_M_nMC_Brake_nValue), 
				BufLen:= SIZEOF(FB_MC2_AX8000_M_nMC_Brake_nValue), 
				Execute:= TRUE, 
				Timeout:= , 
				CompleteAccess:= , 
				Axis:= _stAXIS_REF, 
				Busy=> , 
				Error=> , 
				AdsErrId=> , 
				CANopenErrId=> );	
				
			FB_MC2_AX8000_M_nMC_Brake_iState:= FB_MC2_AX8000_M_nMC_Brake_iState +1;

	003:	// Write brake state
			M_nMC_Brake:= Tc3_HBI_System.cRUNNING;
			FB_MC2_AX8000_M_nMC_Brake_fbCoEWrite(Execute:= TRUE, Axis:= _stAXIS_REF); 
			
			// Error handling
			IF FB_MC2_AX8000_M_nMC_Brake_fbCoEWrite.Error THEN
				M_nError(FB_MC2_AX8000_M_nMC_Brake_fbCoEWrite.AdsErrId);
				M_nMC_Brake:= FB_MC2_AX8000_M_nMC_Brake_fbCoEWrite.AdsErrId;
			ELSE
				// Done
				IF NOT FB_MC2_AX8000_M_nMC_Brake_fbCoEWrite.Busy THEN
					FB_MC2_AX8000_M_nMC_Brake_fbCoEWrite(Execute:= FALSE, Axis:= _stAXIS_REF); 
					FB_MC2_AX8000_M_nMC_Brake_iState:= FB_MC2_AX8000_M_nMC_Brake_iState +1;
				END_IF	
			END_IF
		
	004:	// Done
			M_nMC_Brake:= Tc3_HBI_System.cCOMPLETE;
			IF NOT FB_MC2_AX8000_M_nMC_Brake_bExecute THEN
				FB_MC2_AX8000_M_nMC_Brake_iState:= 000;
			END_IF
			
ELSE
	FB_MC2_AX8000_M_nMC_Brake_iState:= 000;
END_CASE
END_METHOD

//	The result of the method is an unsigned double integer
//	0 = idle 
//	1 = coupled
//	2 = starting
//	3 = running
//	4 = aborted
// 	5 = no hardware connected
// 	6 = Spare
//	7 = pointer or index error
//	8 = mapping error
//	9 = parameter error
//	10 = complete
//	Any other number = ErrorID
METHOD PRIVATE M_nMC_DriveData : UDINT
//**********************************
// Reset 
//**********************************
IF _bReset THEN
	IF _bError THEN
		FB_MC2_AX8000_M_nMC_DriveData_fbCoERead(Execute:= FALSE, Axis:= _stAXIS_REF); 
		FB_MC2_AX8000_M_nMC_DriveData_fbCoEWrite(Execute:= FALSE, Axis:= _stAXIS_REF);
	END_IF
	RETURN;
END_IF

// No hardware connected
IF NOT _bHardwareConnected THEN
	FB_MC2_AX8000_M_nMC_DriveData_lrActualMainVoltage:= 0.0;				// Drive Main voltage
	FB_MC2_AX8000_M_nMC_DriveData_lrAmplifierTemperature:= 0.0;				// Drive temperatur
	FB_MC2_AX8000_M_nMC_DriveData_lrMotorTemperature:= 0.0;					// Motor temperatur
	FB_MC2_AX8000_M_nMC_DriveData_fbCoERead(Execute:= FALSE, Axis:= _stAXIS_REF); 
	FB_MC2_AX8000_M_nMC_DriveData_fbCoEWrite(Execute:= FALSE, Axis:= _stAXIS_REF);
	FB_MC2_AX8000_M_nMC_DriveData_iState:= 000;
	M_nMC_DriveData:= Tc3_HBI_System.cNO_HARDWARE_CONNECTED;
	RETURN;
END_IF


//**********************************
// Main sequence
//**********************************

CASE FB_MC2_AX8000_M_nMC_DriveData_iState OF
	
	000:	// Init
			FB_MC2_AX8000_M_nMC_DriveData_fbCoERead(Execute:= FALSE, Axis:= _stAXIS_REF); 
			FB_MC2_AX8000_M_nMC_DriveData_fbCoEWrite(Execute:= FALSE, Axis:= _stAXIS_REF);
			FB_MC2_AX8000_M_nMC_DriveData_iValue:= 0;
			FB_MC2_AX8000_M_nMC_DriveData_rValue:= 0.0;
			M_nMC_DriveData:= Tc3_HBI_System.cSTARTING;

			// Simulations axis 
			IF _stAXIS_REF.NcToPlc.AxisID > 0 THEN
				IF _stAXIS_REF.Status.OpMode.SimulationAxis THEN
					FB_MC2_AX8000_M_nMC_DriveData_lrActualMainVoltage:= 0.0;			// Drive Main voltage
					FB_MC2_AX8000_M_nMC_DriveData_lrAmplifierTemperature:= 0.0;			// Drive temperatur
					FB_MC2_AX8000_M_nMC_DriveData_lrMotorTemperature:= 0.0;				// Motor temperatur
					M_nMC_DriveData:= Tc3_HBI_System.cNO_HARDWARE_CONNECTED;
				ELSE
					// Axis connected to Hardware
					IF _bHardwareConnected THEN
						M_nMC_DriveData:= Tc3_HBI_System.cCOMPLETE;
						FB_MC2_AX8000_M_nMC_DriveData_iState:= FB_MC2_AX8000_M_nMC_DriveData_iState +1;
					ELSE
						FB_MC2_AX8000_M_nMC_DriveData_lrActualMainVoltage:= 0.0;		// Drive Main voltage
						FB_MC2_AX8000_M_nMC_DriveData_lrAmplifierTemperature:= 0.0;		// Drive temperatur
						FB_MC2_AX8000_M_nMC_DriveData_lrMotorTemperature:= 0.0;			// Motor temperatur
						M_nMC_DriveData:= Tc3_HBI_System.cNO_HARDWARE_CONNECTED;
					END_IF
				END_IF
			ELSE
				FB_MC2_AX8000_M_nMC_DriveData_lrActualMainVoltage:= 0.0;				// Drive Main voltage
				FB_MC2_AX8000_M_nMC_DriveData_lrAmplifierTemperature:= 0.0;				// Drive temperatur
				FB_MC2_AX8000_M_nMC_DriveData_lrMotorTemperature:= 0.0;					// Motor temperatur
				M_nMC_DriveData:= Tc3_HBI_System.cNO_HARDWARE_CONNECTED;
			END_IF
	
//**************************************************************************
// Init values
//**************************************************************************

	001:	// Set motor temp type - 0x32C0:0F
			M_nMC_DriveData:= Tc3_HBI_System.cRUNNING;
			FB_MC2_AX8000_M_nMC_DriveData_iValue:= 1;
			FB_MC2_AX8000_M_nMC_DriveData_fbCoEWrite(
				NetId:= '', 
				Index:= 16#32C0 + (16#0400 * _stDriveAddress.Channel), 
				SubIndex:= 16#0F, 
				pSrcBuf:= ADR(FB_MC2_AX8000_M_nMC_DriveData_iValue), 
				BufLen:= SIZEOF(FB_MC2_AX8000_M_nMC_DriveData_iValue), 
				Execute:= TRUE, 
				Timeout:= , 
				CompleteAccess:= , 
				Axis:= _stAXIS_REF, 
				Busy=> , 
				Error=> , 
				AdsErrId=> , 
				CANopenErrId=> );	

			// Error handling
			IF FB_MC2_AX8000_M_nMC_DriveData_fbCoEWrite.Error THEN
				M_nError(FB_MC2_AX8000_M_nMC_DriveData_fbCoEWrite.AdsErrId);
				M_nMC_DriveData:= FB_MC2_AX8000_M_nMC_DriveData_fbCoEWrite.AdsErrId;
			ELSE
				// Done
				IF NOT FB_MC2_AX8000_M_nMC_DriveData_fbCoEWrite.Busy THEN
					FB_MC2_AX8000_M_nMC_DriveData_fbCoEWrite(Execute:= FALSE, Axis:= _stAXIS_REF);
					FB_MC2_AX8000_M_nMC_DriveData_iValue:= 0;
					FB_MC2_AX8000_M_nMC_DriveData_iState:= 010;
				END_IF
			END_IF
			
//**************************************************************************
// Running values
//**************************************************************************

	010:	// Read motor temp - 0x32C1:06			
			M_nMC_DriveData:= Tc3_HBI_System.cCOMPLETE;
			FB_MC2_AX8000_M_nMC_DriveData_fbCoERead(
				NetId:= '', 
				Index:= 16#32C1 + (16#0400 * _stDriveAddress.Channel), 
				SubIndex:= 16#06, 
				pDstBuf:= ADR(FB_MC2_AX8000_M_nMC_DriveData_rValue), 
				BufLen:= SIZEOF(FB_MC2_AX8000_M_nMC_DriveData_rValue), 
				Execute:= TRUE, 
				Timeout:= , 
				CompleteAccess:= , 
				Axis:= _stAXIS_REF, 
				Busy=> , 
				Error=> , 
				AdsErrId=> , 
				CANopenErrId=> );
		
			// Error handling
			IF FB_MC2_AX8000_M_nMC_DriveData_fbCoERead.Error THEN
				M_nError(FB_MC2_AX8000_M_nMC_DriveData_fbCoERead.AdsErrId);
				M_nMC_DriveData:= FB_MC2_AX8000_M_nMC_DriveData_fbCoERead.AdsErrId;
			ELSE
				// Done
				IF NOT FB_MC2_AX8000_M_nMC_DriveData_fbCoERead.Busy THEN
					FB_MC2_AX8000_M_nMC_DriveData_lrMotorTemperature:= REAL_TO_LREAL(FB_MC2_AX8000_M_nMC_DriveData_rValue);
					FB_MC2_AX8000_M_nMC_DriveData_fbCoERead(Execute:= FALSE, Axis:= _stAXIS_REF);
					FB_MC2_AX8000_M_nMC_DriveData_rValue:= 0.0;
					FB_MC2_AX8000_M_nMC_DriveData_iState:= FB_MC2_AX8000_M_nMC_DriveData_iState +1;
				END_IF
			END_IF

	011:	// Read IGBT temp - 0x3001:02			
			M_nMC_DriveData:= Tc3_HBI_System.cCOMPLETE;
			FB_MC2_AX8000_M_nMC_DriveData_fbCoERead(
				NetId:= '', 
				Index:= 16#3001 + (16#0400 * _stDriveAddress.Channel), 
				SubIndex:= 16#02, 
				pDstBuf:= ADR(FB_MC2_AX8000_M_nMC_DriveData_iValue), 
				BufLen:= SIZEOF(FB_MC2_AX8000_M_nMC_DriveData_iValue), 
				Execute:= TRUE, 
				Timeout:= , 
				CompleteAccess:= , 
				Axis:= _stAXIS_REF, 
				Busy=> , 
				Error=> , 
				AdsErrId=> , 
				CANopenErrId=> );
		
			// Error handling
			IF FB_MC2_AX8000_M_nMC_DriveData_fbCoERead.Error THEN
				M_nError(FB_MC2_AX8000_M_nMC_DriveData_fbCoERead.AdsErrId);
				M_nMC_DriveData:= FB_MC2_AX8000_M_nMC_DriveData_fbCoERead.AdsErrId;
			ELSE
				// Done
				IF NOT FB_MC2_AX8000_M_nMC_DriveData_fbCoERead.Busy THEN
					FB_MC2_AX8000_M_nMC_DriveData_lrAmplifierTemperature:= INT_TO_LREAL(FB_MC2_AX8000_M_nMC_DriveData_iValue);
					FB_MC2_AX8000_M_nMC_DriveData_fbCoERead(Execute:= FALSE, Axis:= _stAXIS_REF);
					FB_MC2_AX8000_M_nMC_DriveData_iValue:= 0;
					FB_MC2_AX8000_M_nMC_DriveData_iState:= FB_MC2_AX8000_M_nMC_DriveData_iState +1;
				END_IF
			END_IF

			
	012:	//
			FB_MC2_AX8000_M_nMC_DriveData_iState:= 010;
	
			
ELSE
	FB_MC2_AX8000_M_nMC_DriveData_iState:= 000;
END_CASE
END_METHOD

//	The result of the method is an unsigned double integer
//	0 = idle 
//	1 = coupled
//	2 = starting
//	3 = running
//	4 = aborted
// 	5 = no hardware connected
// 	6 = Spare
//	7 = pointer or index error
//	8 = mapping error
//	9 = parameter error
//	10 = complete
//	Any other number = ErrorID
METHOD PUBLIC M_nMC_Power : UDINT
VAR_INPUT
	bEnable: BOOL;
	bE_Stop: BOOL;
	bE_StopDelay: BOOL;
	bEnable_Positive: BOOL;
	bEnable_Negative: BOOL;
END_VAR
// Local variable
FB_MC2_AX8000_M_nMC_Power_bEnable:= bEnable;
FB_MC2_AX8000_M_nMC_Power_bE_Stop:= bE_Stop;
FB_MC2_AX8000_M_nMC_Power_bE_StopDelay:= bE_StopDelay; 
FB_MC2_AX8000_M_nMC_Power_bEnable_Positive:= bEnable_Positive;
FB_MC2_AX8000_M_nMC_Power_bEnable_Negative:= bEnable_Negative;

//**********************************
// Reset 
//**********************************
IF _bReset THEN
	MEMSET(destAddr:= ADR(FB_MC2_AX8000_M_nMC_Power_arr_nRet), fillByte:= 16#00, n:= SIZEOF(FB_MC2_AX8000_M_nMC_Power_arr_nRet));
	
	M_nMC_Brake(bExecute:= FB_MC2_AX8000_M_nMC_Brake_bExecute, eBrakeState:= FB_MC2_AX8000_M_nMC_Brake_eBrakeState);
	M_nMC_DriveData();
	M_nMC_Torque(bExecute:= FB_MC2_AX8000_M_nMC_Torque_bExecute, lrTorque:= FB_MC2_AX8000_M_nMC_Torque_lrTorque);
END_IF


//**********************************
// Call methods 
//**********************************
FB_MC2_AX8000_M_nMC_Power_fbStartDelay_TON(IN:= TRUE, PT:= T#200MS, Q=> , ET=> );
IF FB_MC2_AX8000_M_nMC_Power_fbStartDelay_TON.Q THEN
	IF _stAXIS_REF.NcToPlc.AxisID > 0 THEN
		FB_MC2_AX8000_M_nMC_Power_arr_nRet[1]:= SUPER^.M_nMC_Power(bEnable:= FB_MC2_AX8000_M_nMC_Power_bEnable, bE_Stop:= FB_MC2_AX8000_M_nMC_Power_bE_Stop, bE_StopDelay:= FB_MC2_AX8000_M_nMC_Power_bE_StopDelay, bEnable_Positive:= FB_MC2_AX8000_M_nMC_Power_bEnable_Positive, bEnable_Negative:= FB_MC2_AX8000_M_nMC_Power_bEnable_Negative);
		FB_MC2_AX8000_M_nMC_Power_arr_nRet[2]:= M_nMC_DriveData();				
	ELSE
		SUPER^.M_nMC_Power(bEnable:= FALSE, bE_Stop:= FB_MC2_AX8000_M_nMC_Power_bE_Stop, bE_StopDelay:= FB_MC2_AX8000_M_nMC_Power_bE_StopDelay, bEnable_Positive:= FB_MC2_AX8000_M_nMC_Power_bEnable_Positive, bEnable_Negative:= FB_MC2_AX8000_M_nMC_Power_bEnable_Negative);
		IF FB_MC2_AX8000_M_nMC_Power_bEnable THEN
			M_nMC_Power:= Tc3_HBI_System.cMAPPING_ERROR;
		END_IF
		RETURN;
	END_IF
END_IF


//**********************************
// Error handling
//**********************************
IF _stAXIS_REF.Status.Error THEN
	M_nError(_stAXIS_REF.Status.ErrorID);
	M_nMC_Power:= _nErrorID;
ELSE
	FOR _iIdx:= 1 TO UINT_TO_INT(SIZEOF(FB_MC2_AX8000_M_nMC_Power_arr_nRet) / SIZEOF(FB_MC2_AX8000_M_nMC_Power_arr_nRet[1])) DO
		IF FB_MC2_AX8000_M_nMC_Power_arr_nRet[_iIdx] > 5 AND FB_MC2_AX8000_M_nMC_Power_arr_nRet[_iIdx] <> 10 THEN
			M_nError(nErrorID:= FB_MC2_AX8000_M_nMC_Power_arr_nRet[_iIdx]);
			EXIT;
		END_IF
	END_FOR

	// Method return value
	IF _bError THEN
		M_nMC_Power:= _nErrorID;
	ELSE
		M_nMC_Power:= FB_MC2_AX8000_M_nMC_Power_arr_nRet[1];
	END_IF

END_IF
END_METHOD

//	The result of the method is an unsigned double integer
//	0 = idle 
//	1 = coupled
//	2 = starting
//	3 = running
//	4 = aborted
// 	5 = no hardware connected
// 	6 = Spare
//	7 = pointer or index error
//	8 = mapping error
//	9 = parameter error
//	10 = complete
//	Any other number = ErrorID
METHOD PUBLIC M_nMC_Torque : UDINT
VAR_INPUT
	bExecute: BOOL;
	lrTorque: LREAL; 		// Torque limit 0.0-500.0%	
END_VAR
// Local variable
FB_MC2_AX8000_M_nMC_Torque_bExecute:= bExecute;
FB_MC2_AX8000_M_nMC_Torque_lrTorque:= lrTorque;

//**********************************
// Reset 
//**********************************
IF _bReset THEN
	IF _bError THEN
		FB_MC2_AX8000_M_nMC_Torque_fbCoEWrite(Execute:= FALSE, Axis:= _stAXIS_REF); 
		FB_MC2_AX8000_M_nMC_Torque_fbExecute_R_TRIG(CLK:= FALSE);
		FB_MC2_AX8000_M_nMC_Torque_iState:= 000;
	END_IF
END_IF
// No hardware connected
IF NOT _bHardwareConnected THEN
	FB_MC2_AX8000_M_nMC_Torque_fbCoEWrite(Execute:= FALSE, Axis:= _stAXIS_REF); 
	FB_MC2_AX8000_M_nMC_Torque_fbExecute_R_TRIG(CLK:= FALSE);
	FB_MC2_AX8000_M_nMC_Torque_iState:= 000;
	IF FB_MC2_AX8000_M_nMC_Torque_bExecute THEN
		M_nMC_Torque:= Tc3_HBI_System.cNO_HARDWARE_CONNECTED;
	END_IF		
	RETURN;
END_IF

//**********************************
// Parameter check 
//**********************************
IF FB_MC2_AX8000_M_nMC_Torque_bExecute THEN
	IF FB_MC2_AX8000_M_nMC_Torque_lrTorque < 0.0 OR FB_MC2_AX8000_M_nMC_Torque_lrTorque > 500.0 THEN
		M_nMC_Torque:= Tc3_HBI_System.cPARAMETER_ERROR;
		
		FB_MC2_AX8000_M_nMC_Torque_fbCoEWrite(Execute:= FALSE, Axis:= _stAXIS_REF); 
		FB_MC2_AX8000_M_nMC_Torque_fbExecute_R_TRIG(CLK:= FALSE);
		FB_MC2_AX8000_M_nMC_Torque_iState:= 000;
		RETURN;
	END_IF
END_IF


//**********************************
// Wait for execute
//**********************************
IF _stAXIS_REF.NcToPlc.AxisID > 0 THEN
	FB_MC2_AX8000_M_nMC_Torque_fbExecute_R_TRIG(CLK:= FB_MC2_AX8000_M_nMC_Torque_bExecute);
	IF FB_MC2_AX8000_M_nMC_Torque_fbExecute_R_TRIG.Q THEN
		FB_MC2_AX8000_M_nMC_Torque_fbCoEWrite(Execute:= FALSE, Axis:= _stAXIS_REF); 
		FB_MC2_AX8000_M_nMC_Torque_iState:= 001;
	END_IF
ELSE
	FB_MC2_AX8000_M_nMC_Torque_fbExecute_R_TRIG(CLK:= FALSE);
	FB_MC2_AX8000_M_nMC_Torque_iState:= 000;
	IF FB_MC2_AX8000_M_nMC_Torque_bExecute THEN
		M_nMC_Torque:= Tc3_HBI_System.cMAPPING_ERROR;
	END_IF
	RETURN;
END_IF


//**********************************
// Main sequence
//**********************************
CASE FB_MC2_AX8000_M_nMC_Torque_iState OF

	000: 	// Do nothing
	
	001:	// Write torque limet	
			M_nMC_Torque:= Tc3_HBI_System.cRUNNING;
			FB_MC2_AX8000_M_nMC_Torque_iTorque:= LREAL_TO_INT(FB_MC2_AX8000_M_nMC_Torque_lrTorque * 10);
			FB_MC2_AX8000_M_nMC_Torque_fbCoEWrite(
				NetId:= '', 
				Index:= 16#6072 + (16#0800 * _stDriveAddress.Channel), 
				SubIndex:= 16#00, 
				pSrcBuf:= ADR(FB_MC2_AX8000_M_nMC_Torque_iTorque), 
				BufLen:= SIZEOF(FB_MC2_AX8000_M_nMC_Torque_iTorque), 
				Execute:= TRUE, 
				Timeout:= , 
				CompleteAccess:= , 
				Axis:= _stAXIS_REF, 
				Busy=> , 
				Error=> , 
				AdsErrId=> , 
				CANopenErrId=> );	
			
			FB_MC2_AX8000_M_nMC_Torque_iState:= FB_MC2_AX8000_M_nMC_Torque_iState +1;
			
	002:	// Write torque limet
			M_nMC_Torque:= Tc3_HBI_System.cRUNNING;
			FB_MC2_AX8000_M_nMC_Torque_fbCoEWrite(Execute:= TRUE, Axis:= _stAXIS_REF); 
			
			// Error handling
			IF FB_MC2_AX8000_M_nMC_DriveData_fbCoEWrite.Error THEN
				M_nError(FB_MC2_AX8000_M_nMC_DriveData_fbCoEWrite.AdsErrId);
				M_nMC_Torque:= FB_MC2_AX8000_M_nMC_DriveData_fbCoEWrite.AdsErrId;
			ELSE
				// Done
				IF NOT FB_MC2_AX8000_M_nMC_Torque_fbCoEWrite.Busy THEN
					FB_MC2_AX8000_M_nMC_Torque_fbCoEWrite(Execute:= FALSE, Axis:= _stAXIS_REF); 
					FB_MC2_AX8000_M_nMC_Torque_iState:= FB_MC2_AX8000_M_nMC_Torque_iState +1;
				END_IF	
			END_IF
		
	003:	// Done
			M_nMC_Torque:= Tc3_HBI_System.cCOMPLETE;
			IF NOT FB_MC2_AX8000_M_nMC_Torque_bExecute THEN
				FB_MC2_AX8000_M_nMC_Torque_iState:= 000;
			END_IF
		
ELSE
	FB_MC2_AX8000_M_nMC_Torque_iState:= 000;
END_CASE
END_METHOD

//	The result of the method is an unsigned double integer
//	0 = idle 
//	1 = coupled
//	2 = starting
//	3 = running
//	4 = aborted
// 	5 = no hardware connected
// 	6 = Spare
//	7 = pointer or index error
//	8 = mapping error
//	9 = parameter error
//	10 = complete
//	Any other number = ErrorID
METHOD PUBLIC M_nReset : UDINT
VAR_INPUT
	bExecute: BOOL;
END_VAR
//**********************************
// Wait for execute
//**********************************
FB_MC2_AX8000_M_nReset_fbExecute_R_TRIG(CLK:= bExecute);
IF FB_MC2_AX8000_M_nReset_fbExecute_R_TRIG.Q THEN
	SUPER^.M_nReset(bExecute:= FALSE);
	FB_MC2_AX8000_M_nReset_iState:= 001;
END_IF


//**********************************
// Main sequence
//**********************************
CASE FB_MC2_AX8000_M_nReset_iState OF

	000: 	// Do nothing

	001:	// Reset father	
			M_nReset:= Tc3_HBI_System.cRUNNING;
			FB_MC2_AX8000_M_nReset_nStatus:= SUPER^.M_nReset(bExecute:= TRUE); 
			IF FB_MC2_AX8000_M_nReset_nStatus = Tc3_HBI_System.cCOUPLED OR FB_MC2_AX8000_M_nReset_nStatus = Tc3_HBI_System.cCOMPLETE THEN		
				SUPER^.M_nReset(bExecute:= FALSE);
				IF _stAXIS_REF.Status.Coupled THEN
					FB_MC2_AX8000_M_nReset_iState:= 020;
				ELSE
					FB_MC2_AX8000_M_nReset_iState:= 030;
				END_IF
			END_IF

	020:	// Coupled
			M_nReset:= Tc3_HBI_System.cCOUPLED;
			IF NOT bExecute THEN
				SUPER^.M_nReset(bExecute:= FALSE);
				FB_MC2_AX8000_M_nReset_iState:= 000;
			END_IF	

	030: 	// Done
			M_nReset:= Tc3_HBI_System.cCOMPLETE;
			IF NOT bExecute THEN
				SUPER^.M_nReset(bExecute:= FALSE);
				FB_MC2_AX8000_M_nReset_iState:= 000;
			END_IF	
		
ELSE
	FB_MC2_AX8000_M_nReset_iState:= 000;
END_CASE
END_METHOD

PROPERTY PUBLIC P_rActualMainVoltage : REAL
GET
P_rActualMainVoltage:= LREAL_TO_REAL(FB_MC2_AX8000_M_nMC_DriveData_lrActualMainVoltage);
END_GET
END_PROPERTY

PROPERTY PUBLIC P_rAmplifierTemperature : REAL
GET
P_rAmplifierTemperature:= LREAL_TO_REAL(FB_MC2_AX8000_M_nMC_DriveData_lrAmplifierTemperature);
END_GET
END_PROPERTY

PROPERTY PUBLIC P_rMotorTemperature : REAL
GET
P_rMotorTemperature:= LREAL_TO_REAL(FB_MC2_AX8000_M_nMC_DriveData_lrMotorTemperature);
END_GET
END_PROPERTY

END_FUNCTION_BLOCK

// MOTION/POUs/FBs/Basic/FB_MC2_EL70xx
//------------------------------------------------------------------------------------------
//                                                                                        	
//***************************** Beckhoff TwinCAT Examples **********************************
//                                                                                        	
//************************************* WARNING ********************************************
// This program is only an example. If it is used as a control program in any real        	
// application, Beckhoff is not responsible for any malfunction, loss or damage           	
// which could arise by using this program!                                               	
//                                                                                        	
//*************************************  Program Info. *************************************
//                                                                                        	
// PLC program name:      	FB_MC2_Stepper (FB)                                          	
// Hardware platform:      	TwinCat PTP v3.1.4022				                          		                                  	
//                                                                                        	
// ======================================================================================== 
//         Version       Date                        Remarks                              	
// ======================================================================================== 
//         3.1           27 feb 2018                 First release of this example        	
// ======================================================================================== 
//                                                                                        	
//******************************* Aims OF this PLC PROGRAM *********************************
//                                                                                        	
// MC2 stepper servo axis 						 			                                      	
//																	                      	
//                                                                                        	
//----------------------------------------------------------------------------------------- 
FUNCTION_BLOCK FB_MC2_EL70xx EXTENDS FB_MC2_Basic IMPLEMENTS I_MC2_EL70xx
VAR
//********************************
// Methods variable
//********************************
	FB_MC2_EL70xx_M_nMC_DriveData_iState: INT;
	FB_MC2_EL70xx_M_nMC_DriveData_fbEcCoESdoRead: FB_EcCoESdoRead;
	FB_MC2_EL70xx_M_nMC_DriveData_fbDelay_TON: TC2_STANDARD.TON;
	FB_MC2_EL70xx_M_nMC_DriveData_nByte: BYTE;
	FB_MC2_EL70xx_M_nMC_DriveData_nDInt: DINT;
	FB_MC2_EL70xx_M_nMC_DriveData_lrControlVoltage: LREAL;
	FB_MC2_EL70xx_M_nMC_DriveData_lrAmplifierTemperature: LREAL;
	FB_MC2_EL70xx_M_nMC_DriveData_lrMotorSupplyVoltage: LREAL;

	FB_MC2_EL70xx_M_nMC_Power_bEnable: BOOL;
	FB_MC2_EL70xx_M_nMC_Power_bE_Stop: BOOL;
	FB_MC2_EL70xx_M_nMC_Power_bE_StopDelay: BOOL;
	FB_MC2_EL70xx_M_nMC_Power_bEnable_Positive: BOOL;
	FB_MC2_EL70xx_M_nMC_Power_bEnable_Negative: BOOL;
	FB_MC2_EL70xx_M_nMC_Power_fbStartDelay_TON: Tc2_Standard.TON;
	FB_MC2_EL70xx_M_nMC_Power_arr_nRet: ARRAY[1..3] OF UDINT;
END_VAR

//	The result of the method is an unsigned double integer
//	0 = idle 
//	1 = coupled
//	2 = starting
//	3 = running
//	4 = aborted
// 	5 = no hardware connected
// 	6 = Spare
//	7 = pointer or index error
//	8 = mapping error
//	9 = parameter error
//	10 = complete
//	Any other number = ErrorID
METHOD PRIVATE M_nMC_DriveData : UDINT
//**********************************
// Reset 
//**********************************
IF _bReset THEN
	IF _bError THEN
		FB_MC2_EL70xx_M_nMC_DriveData_iState:= 000;
	END_IF
END_IF

// No hardware connected
IF NOT _bHardwareConnected THEN
	FB_MC2_EL70xx_M_nMC_DriveData_lrAmplifierTemperature:= 0.0;			// Terminal intern temperatur
	FB_MC2_EL70xx_M_nMC_DriveData_lrControlVoltage:= 0.0;				// Control voltage 24v
	FB_MC2_EL70xx_M_nMC_DriveData_lrMotorSupplyVoltage:= 0.0;			// Motor voltage
	FB_MC2_EL70xx_M_nMC_DriveData_iState:= 000;
	M_nMC_DriveData:= Tc3_HBI_System.cNO_HARDWARE_CONNECTED;
	RETURN;
END_IF

// Check for Axis
IF _stAXIS_REF.NcToPlc.AxisID = 0 THEN
	FB_MC2_EL70xx_M_nMC_DriveData_iState:= 000;
	RETURN;
END_IF


// Main sequence
CASE FB_MC2_EL70xx_M_nMC_DriveData_iState OF

	000: 	// Init
			M_nMC_DriveData:= Tc3_HBI_System.cSTARTING;
			FB_MC2_EL70xx_M_nMC_DriveData_fbEcCoESdoRead(bExecute:= FALSE);
	
			IF _stAXIS_REF.NcToPlc.AxisID > 0 THEN
				// Simulations axis 
				IF NOT _stAXIS_REF.Status.OpMode.SimulationAxis THEN
					FB_MC2_EL70xx_M_nMC_DriveData_lrAmplifierTemperature:= 0.0;				// Terminal intern temperatur
					FB_MC2_EL70xx_M_nMC_DriveData_lrControlVoltage:= 0.0;					// Control voltage 24v
					FB_MC2_EL70xx_M_nMC_DriveData_lrMotorSupplyVoltage:= 0.0;				// Motor voltage
					M_nMC_DriveData:= Tc3_HBI_System.cNO_HARDWARE_CONNECTED;
				ELSE
					// Axis connected to Hardware
					IF _bHardwareConnected THEN
						M_nMC_DriveData:= Tc3_HBI_System.cCOMPLETE;
						FB_MC2_EL70xx_M_nMC_DriveData_iState:= FB_MC2_EL70xx_M_nMC_DriveData_iState +1;
					ELSE
						FB_MC2_EL70xx_M_nMC_DriveData_lrAmplifierTemperature:= 0.0;			// Terminal intern temperatur
						FB_MC2_EL70xx_M_nMC_DriveData_lrControlVoltage:= 0.0;				// Control voltage 24v
						FB_MC2_EL70xx_M_nMC_DriveData_lrMotorSupplyVoltage:= 0.0;			// Motor voltage
						M_nMC_DriveData:= Tc3_HBI_System.cNO_HARDWARE_CONNECTED;
					END_IF
				END_IF
			ELSE
				FB_MC2_EL70xx_M_nMC_DriveData_lrAmplifierTemperature:= 0.0;			// Terminal intern temperatur
				FB_MC2_EL70xx_M_nMC_DriveData_lrControlVoltage:= 0.0;				// Control voltage 24v
				FB_MC2_EL70xx_M_nMC_DriveData_lrMotorSupplyVoltage:= 0.0;			// Motor voltage
				M_nMC_DriveData:= Tc3_HBI_System.cNO_HARDWARE_CONNECTED;
			END_IF
		
	001:	// Read Internal temperatur 
			M_nMC_DriveData:= Tc3_HBI_System.cCOMPLETE;
			FB_MC2_EL70xx_M_nMC_DriveData_fbEcCoESdoRead(bExecute:= FALSE);
			FB_MC2_EL70xx_M_nMC_DriveData_fbEcCoESdoRead(
				sNetId:= _stDriveAddress.NetID, 
				nSlaveAddr:= _stDriveAddress.SlaveAddress, 
				nSubIndex:= 16#02, 
				nIndex:= 16#F900, 
				pDstBuf:= ADR(FB_MC2_EL70xx_M_nMC_DriveData_nByte), 
				cbBufLen:= SIZEOF(FB_MC2_EL70xx_M_nMC_DriveData_nByte), 
				bExecute:= TRUE, 
				tTimeout:= T#2S);
	 
			FB_MC2_EL70xx_M_nMC_DriveData_iState:= FB_MC2_EL70xx_M_nMC_DriveData_iState +1;
	
	002:	// Error handling
			M_nMC_DriveData:= Tc3_HBI_System.cCOMPLETE;
			FB_MC2_EL70xx_M_nMC_DriveData_fbEcCoESdoRead(bExecute:= TRUE);
			IF FB_MC2_EL70xx_M_nMC_DriveData_fbEcCoESdoRead.bError THEN
				M_nError(nErrorID:= FB_MC2_EL70xx_M_nMC_DriveData_fbEcCoESdoRead.nErrId);
				M_nMC_DriveData:= FB_MC2_EL70xx_M_nMC_DriveData_fbEcCoESdoRead.nErrId;
			ELSE
				// Done
				IF NOT FB_MC2_EL70xx_M_nMC_DriveData_fbEcCoESdoRead.bBusy THEN
					FB_MC2_EL70xx_M_nMC_DriveData_fbEcCoESdoRead(bExecute:= FALSE);
					FB_MC2_EL70xx_M_nMC_DriveData_lrAmplifierTemperature:= BYTE_TO_LREAL(FB_MC2_EL70xx_M_nMC_DriveData_nByte);
					FB_MC2_EL70xx_M_nMC_DriveData_iState:= FB_MC2_EL70xx_M_nMC_DriveData_iState +1;
				END_IF	
			END_IF
	
	003:	// Read Control voltage 24v 
			M_nMC_DriveData:= Tc3_HBI_System.cCOMPLETE;
			FB_MC2_EL70xx_M_nMC_DriveData_fbEcCoESdoRead(bExecute:= FALSE);
			FB_MC2_EL70xx_M_nMC_DriveData_fbEcCoESdoRead(
				sNetId:= _stDriveAddress.NetID, 
				nSlaveAddr:= _stDriveAddress.SlaveAddress, 
				nSubIndex:= 16#04, 
				nIndex:= 16#F900, 
				pDstBuf:= ADR(FB_MC2_EL70xx_M_nMC_DriveData_nDInt), 
				cbBufLen:= SIZEOF(FB_MC2_EL70xx_M_nMC_DriveData_nDInt), 
				bExecute:= TRUE, 
				tTimeout:= T#2S);
	 
			FB_MC2_EL70xx_M_nMC_DriveData_iState:= FB_MC2_EL70xx_M_nMC_DriveData_iState +1;

	004:	// Error handling
			M_nMC_DriveData:= Tc3_HBI_System.cCOMPLETE;
			FB_MC2_EL70xx_M_nMC_DriveData_fbEcCoESdoRead(bExecute:= TRUE);
			IF FB_MC2_EL70xx_M_nMC_DriveData_fbEcCoESdoRead.bError THEN
				M_nError(nErrorID:= FB_MC2_EL70xx_M_nMC_DriveData_fbEcCoESdoRead.nErrId);
				M_nMC_DriveData:= FB_MC2_EL70xx_M_nMC_DriveData_fbEcCoESdoRead.nErrId;
			ELSE
				// Done
				IF NOT FB_MC2_EL70xx_M_nMC_DriveData_fbEcCoESdoRead.bBusy THEN
					FB_MC2_EL70xx_M_nMC_DriveData_fbEcCoESdoRead(bExecute:= FALSE);
					FB_MC2_EL70xx_M_nMC_DriveData_lrControlVoltage:= (DINT_TO_LREAL(FB_MC2_EL70xx_M_nMC_DriveData_nDInt)) / 1000.0;
					FB_MC2_EL70xx_M_nMC_DriveData_iState:= FB_MC2_EL70xx_M_nMC_DriveData_iState +1;
				END_IF	
			END_IF
	
	005:	// Read Motor supply voltage 
			M_nMC_DriveData:= Tc3_HBI_System.cCOMPLETE;
			FB_MC2_EL70xx_M_nMC_DriveData_fbEcCoESdoRead(bExecute:= FALSE);
			FB_MC2_EL70xx_M_nMC_DriveData_fbEcCoESdoRead(
				sNetId:= _stDriveAddress.NetID, 
				nSlaveAddr:= _stDriveAddress.SlaveAddress, 
				nSubIndex:= 16#05, 
				nIndex:= 16#F900, 
				pDstBuf:= ADR(FB_MC2_EL70xx_M_nMC_DriveData_nDInt), 
				cbBufLen:= SIZEOF(FB_MC2_EL70xx_M_nMC_DriveData_nDInt), 
				bExecute:= TRUE, 
				tTimeout:= T#2S);
	 
			FB_MC2_EL70xx_M_nMC_DriveData_iState:= FB_MC2_EL70xx_M_nMC_DriveData_iState +1;

	006:	// Error handling
			M_nMC_DriveData:= Tc3_HBI_System.cCOMPLETE;
			FB_MC2_EL70xx_M_nMC_DriveData_fbEcCoESdoRead(bExecute:= TRUE);
			IF FB_MC2_EL70xx_M_nMC_DriveData_fbEcCoESdoRead.bError THEN
				M_nError(nErrorID:= FB_MC2_EL70xx_M_nMC_DriveData_fbEcCoESdoRead.nErrId);
				M_nMC_DriveData:= FB_MC2_EL70xx_M_nMC_DriveData_fbEcCoESdoRead.nErrId; 
			ELSE
				// Done
				IF NOT FB_MC2_EL70xx_M_nMC_DriveData_fbEcCoESdoRead.bBusy THEN
					FB_MC2_EL70xx_M_nMC_DriveData_fbEcCoESdoRead(bExecute:= FALSE);
					FB_MC2_EL70xx_M_nMC_DriveData_lrMotorSupplyVoltage:= (DINT_TO_LREAL(FB_MC2_EL70xx_M_nMC_DriveData_nDInt)) / 1000.0;
					FB_MC2_EL70xx_M_nMC_DriveData_iState:= FB_MC2_EL70xx_M_nMC_DriveData_iState +1;
				END_IF	
			END_IF
		
	007:	// Done		
			M_nMC_DriveData:= Tc3_HBI_System.cCOMPLETE;
			FB_MC2_EL70xx_M_nMC_DriveData_iState:= 000;
	
ELSE
	FB_MC2_EL70xx_M_nMC_DriveData_iState:= 000;
END_CASE
END_METHOD

//	The result of the method is an unsigned double integer
//	0 = idle 
//	1 = coupled
//	2 = starting
//	3 = running
//	4 = aborted
// 	5 = no hardware connected
// 	6 = Spare
//	7 = pointer or index error
//	8 = mapping error
//	9 = parameter error
//	10 = complete
//	Any other number = ErrorID
METHOD PUBLIC M_nMC_Power : UDINT
VAR_INPUT
	bEnable: BOOL;
	bE_Stop: BOOL;
	bE_StopDelay: BOOL;
	bEnable_Positive: BOOL;
	bEnable_Negative: BOOL;
END_VAR
// Local variable
FB_MC2_EL70xx_M_nMC_Power_bEnable:= bEnable;
FB_MC2_EL70xx_M_nMC_Power_bE_Stop:= bE_Stop;
FB_MC2_EL70xx_M_nMC_Power_bE_StopDelay:= bE_StopDelay;
FB_MC2_EL70xx_M_nMC_Power_bEnable_Positive:= bEnable_Positive;
FB_MC2_EL70xx_M_nMC_Power_bEnable_Negative:= bEnable_Negative;

//**********************************
// Reset 
//**********************************
IF _bReset THEN
	MEMSET(destAddr:= ADR(FB_MC2_EL70xx_M_nMC_Power_arr_nRet), fillByte:= 16#00, n:= SIZEOF(FB_MC2_EL70xx_M_nMC_Power_arr_nRet));

	// Reset all methods
	M_nMC_DriveData();
END_IF

//**********************************
// Call methodes				
//**********************************
FB_MC2_EL70xx_M_nMC_Power_fbStartDelay_TON(IN:= TRUE, PT:= T#200MS, Q=> , ET=> );
IF _stAXIS_REF.NcToPlc.AxisID > 0 OR FB_MC2_EL70xx_M_nMC_Power_fbStartDelay_TON.Q THEN
	FB_MC2_EL70xx_M_nMC_Power_arr_nRet[1]:= SUPER^.M_nMC_Power(bEnable:= FB_MC2_EL70xx_M_nMC_Power_bEnable, bE_Stop:= FB_MC2_EL70xx_M_nMC_Power_bE_Stop, bE_StopDelay:= FB_MC2_EL70xx_M_nMC_Power_bE_StopDelay, bEnable_Positive:= FB_MC2_EL70xx_M_nMC_Power_bEnable_Positive, bEnable_Negative:= FB_MC2_EL70xx_M_nMC_Power_bEnable_Negative);
	FB_MC2_EL70xx_M_nMC_Power_arr_nRet[2]:= M_nMC_DriveData();
	FB_MC2_EL70xx_M_nMC_Power_arr_nRet[3]:= M_nMC_DeadTimeComp();
ELSE
	SUPER^.M_nMC_Power(bEnable:= FALSE, bE_Stop:= FB_MC2_EL70xx_M_nMC_Power_bE_Stop, bE_StopDelay:= FB_MC2_EL70xx_M_nMC_Power_bE_StopDelay, bEnable_Positive:= FB_MC2_EL70xx_M_nMC_Power_bEnable_Positive, bEnable_Negative:= FB_MC2_EL70xx_M_nMC_Power_bEnable_Negative);
	IF FB_MC2_EL70xx_M_nMC_Power_bEnable THEN
		M_nMC_Power:= Tc3_HBI_System.cMAPPING_ERROR;
	END_IF
	RETURN;
END_IF


//**********************************
// Error handling
//**********************************
IF _stAXIS_REF.Status.Error THEN
	M_nError(_stAXIS_REF.Status.ErrorID);
	M_nMC_Power:= _nErrorID;
ELSE
	FOR _iIdx:= 1 TO UINT_TO_INT(SIZEOF(FB_MC2_EL70xx_M_nMC_Power_arr_nRet) / SIZEOF(FB_MC2_EL70xx_M_nMC_Power_arr_nRet[1])) DO
		IF FB_MC2_EL70xx_M_nMC_Power_arr_nRet[_iIdx] > 5 AND FB_MC2_EL70xx_M_nMC_Power_arr_nRet[_iIdx] <> 10 THEN
			M_nError(nErrorID:= FB_MC2_EL70xx_M_nMC_Power_arr_nRet[_iIdx]);
			EXIT;
		END_IF
	END_FOR

	// Method return value
	IF _bError THEN
		M_nMC_Power:= _nErrorID;
	ELSE
		M_nMC_Power:= FB_MC2_EL70xx_M_nMC_Power_arr_nRet[1];
	END_IF

END_IF
END_METHOD

PROPERTY PUBLIC P_rAmplifierTemperature : REAL
GET
P_rAmplifierTemperature:= LREAL_TO_REAL(FB_MC2_EL70xx_M_nMC_DriveData_lrAmplifierTemperature);
END_GET
END_PROPERTY

PROPERTY PUBLIC P_rControlVoltage : REAL
GET
P_rControlVoltage:= LREAL_TO_REAL(FB_MC2_EL70xx_M_nMC_DriveData_lrControlVoltage);
END_GET
END_PROPERTY

PROPERTY PUBLIC P_rMotorSupplyVoltage : REAL
GET
P_rMotorSupplyVoltage:= LREAL_TO_REAL(FB_MC2_EL70xx_M_nMC_DriveData_lrMotorSupplyVoltage);
END_GET
END_PROPERTY

END_FUNCTION_BLOCK

// MOTION/POUs/FBs/Basic/FB_MC2_EL72xx
//------------------------------------------------------------------------------------------
//                                                                                        	
//***************************** Beckhoff TwinCAT Examples **********************************
//                                                                                        	
//************************************* WARNING ********************************************
// This program is only an example. If it is used as a control program in any real        	
// application, Beckhoff is not responsible for any malfunction, loss or damage           	
// which could arise by using this program!                                               	
//                                                                                        	
//*************************************  Program Info. *************************************
//                                                                                        	
// PLC program name:       	FB_MC2_EL7201 (FB)                                          	
// Hardware platform:      	TwinCat PTP v3.1.4022				                          	                                 	
//                                                                                        	
// ======================================================================================== 
//         Version       Date                        Remarks                              	
// ======================================================================================== 
//         3.1           27 feb 2018                 First release of this example        	
// ======================================================================================== 
//                                                                                        	
//******************************* Aims OF this PLC PROGRAM *********************************
//                                                                                        	
// MC2 terminal servo axis 						 			                                      	
//																	                      	
//                                                                                        	
//----------------------------------------------------------------------------------------- 
FUNCTION_BLOCK FB_MC2_EL72xx EXTENDS FB_MC2_Basic IMPLEMENTS I_MC2_EL72xx
VAR
//********************************
// Methods variable
//********************************
	FB_MC2_EL72xx_M_nMC_DriveData_bMDP742: BOOL;
	FB_MC2_EL72xx_M_nMC_DriveData_bDS402: BOOL;
	FB_MC2_EL72xx_M_nMC_DriveData_iState: INT;
	FB_MC2_EL72xx_M_nMC_DriveData_fbEcCoESdoRead: FB_EcCoESdoRead;
	FB_MC2_EL72xx_M_nMC_DriveData_nInt: UINT;
	FB_MC2_EL72xx_M_nMC_DriveData_nDInt: DINT;
	FB_MC2_EL72xx_M_nMC_DriveData_lrAmplifierTemperature: LREAL;
	FB_MC2_EL72xx_M_nMC_DriveData_lrMotorSupplyVoltage: LREAL;
	FB_MC2_EL72xx_M_nMC_DriveData_lrMotorTemperature: LREAL;
	
	FB_MC2_EL72xx_M_nMC_Power_bEnable: BOOL;
	FB_MC2_EL72xx_M_nMC_Power_bE_Stop: BOOL;
	FB_MC2_EL72xx_M_nMC_Power_bE_StopDelay: BOOL;
	FB_MC2_EL72xx_M_nMC_Power_bEnable_Positive: BOOL;
	FB_MC2_EL72xx_M_nMC_Power_bEnable_Negative: BOOL;
	FB_MC2_EL72xx_M_nMC_Power_fbStartDelay_TON: Tc2_Standard.TON;
	FB_MC2_EL72xx_M_nMC_Power_arr_nRet: ARRAY[1..3] OF UDINT;
END_VAR

//	The result of the method is an unsigned double integer
//	0 = idle 
//	1 = coupled
//	2 = starting
//	3 = running
//	4 = aborted
// 	5 = no hardware connected
// 	6 = Spare
//	7 = pointer or index error
//	8 = mapping error
//	9 = parameter error
//	10 = complete
//	Any other number = ErrorID
METHOD PRIVATE M_nMC_DriveData : UDINT
//**********************************
// Reset 
//**********************************
IF _bReset THEN
	IF _bError THEN
		FB_MC2_EL72xx_M_nMC_DriveData_bMDP742:= FALSE;
		FB_MC2_EL72xx_M_nMC_DriveData_bDS402:= FALSE;
		FB_MC2_EL72xx_M_nMC_DriveData_iState:= 000;
	END_IF
END_IF

// No hardware connected
IF NOT _bHardwareConnected THEN
	FB_MC2_EL72xx_M_nMC_DriveData_lrAmplifierTemperature:= 0.0;			// Terminal intern temperatur
	FB_MC2_EL72xx_M_nMC_DriveData_lrMotorSupplyVoltage:= 0.0;			// Motor voltage
	FB_MC2_EL72xx_M_nMC_DriveData_lrMotorTemperature:= 0.0;				// Motor temperatur
	FB_MC2_EL72xx_M_nMC_DriveData_bMDP742:= FALSE;
	FB_MC2_EL72xx_M_nMC_DriveData_bDS402:= FALSE;
	FB_MC2_EL72xx_M_nMC_DriveData_iState:= 000;
	M_nMC_DriveData:= Tc3_HBI_System.cNO_HARDWARE_CONNECTED;
	RETURN;
END_IF	

// Check for Axis
IF _stAXIS_REF.NcToPlc.AxisID = 0 THEN
	FB_MC2_EL72xx_M_nMC_DriveData_bMDP742:= FALSE;
	FB_MC2_EL72xx_M_nMC_DriveData_bDS402:= FALSE;
	FB_MC2_EL72xx_M_nMC_DriveData_iState:= 000;
	RETURN;
END_IF


//**********************************
// Main sequence
//**********************************
CASE FB_MC2_EL72xx_M_nMC_DriveData_iState OF

	000: 	// Init
			M_nMC_DriveData:= Tc3_HBI_System.cCOMPLETE;
			FB_MC2_EL72xx_M_nMC_DriveData_fbEcCoESdoRead(bExecute:= FALSE);
			
			// Simulations axis 
			IF _stAXIS_REF.NcToPlc.AxisID > 0 THEN
				IF _stAXIS_REF.Status.OpMode.SimulationAxis THEN
					FB_MC2_EL72xx_M_nMC_DriveData_lrAmplifierTemperature:= 0.0;			// Terminal intern temperatur
					FB_MC2_EL72xx_M_nMC_DriveData_lrMotorSupplyVoltage:= 0.0;			// Motor voltage
					FB_MC2_EL72xx_M_nMC_DriveData_lrMotorTemperature:= 0.0;				// Motor temperatur
					M_nMC_DriveData:= Tc3_HBI_System.cNO_HARDWARE_CONNECTED;
				ELSE
					// Axis connected to Hardware
					IF _bHardwareConnected THEN
						M_nMC_DriveData:= Tc3_HBI_System.cCOMPLETE;
						FB_MC2_EL72xx_M_nMC_DriveData_iState:= FB_MC2_EL72xx_M_nMC_DriveData_iState +1;
					ELSE
						FB_MC2_EL72xx_M_nMC_DriveData_lrAmplifierTemperature:= 0.0;		// Terminal intern temperatur
						FB_MC2_EL72xx_M_nMC_DriveData_lrMotorSupplyVoltage:= 0.0;		// Motor voltage
						FB_MC2_EL72xx_M_nMC_DriveData_lrMotorTemperature:= 0.0;			// Motor temperatur
						M_nMC_DriveData:= Tc3_HBI_System.cNO_HARDWARE_CONNECTED;
					END_IF
				END_IF
			ELSE
				FB_MC2_EL72xx_M_nMC_DriveData_lrAmplifierTemperature:= 0.0;			// Terminal intern temperatur
				FB_MC2_EL72xx_M_nMC_DriveData_lrMotorSupplyVoltage:= 0.0;			// Motor voltage
				FB_MC2_EL72xx_M_nMC_DriveData_lrMotorTemperature:= 0.0;				// Motor temperatur
				M_nMC_DriveData:= Tc3_HBI_System.cNO_HARDWARE_CONNECTED;
			END_IF

	001:	// Check for MDP742 or DS402 profile 
			IF FB_MC2_EL72xx_M_nMC_DriveData_bMDP742 THEN
				FB_MC2_EL72xx_M_nMC_DriveData_iState:= 010;
			ELSE
				IF FB_MC2_EL72xx_M_nMC_DriveData_bDS402 THEN
					FB_MC2_EL72xx_M_nMC_DriveData_iState:= 020;
				ELSE
					FB_MC2_EL72xx_M_nMC_DriveData_iState:= FB_MC2_EL72xx_M_nMC_DriveData_iState +1;
				END_IF
			END_IF	

	002:	// Check - MDP742 profile
			M_nMC_DriveData:= Tc3_HBI_System.cRUNNING;
			FB_MC2_EL72xx_M_nMC_DriveData_fbEcCoESdoRead(bExecute:= FALSE);
			FB_MC2_EL72xx_M_nMC_DriveData_fbEcCoESdoRead(
				sNetId:= _stDriveAddress.NetID, 
				nSlaveAddr:= _stDriveAddress.SlaveAddress, 
				nSubIndex:= 16#11, 
				nIndex:= 16#9010, 
				pDstBuf:= ADR(FB_MC2_EL72xx_M_nMC_DriveData_nInt), 
				cbBufLen:= SIZEOF(FB_MC2_EL72xx_M_nMC_DriveData_nInt), 
				bExecute:= TRUE, 
				tTimeout:= T#2S);
	 
			FB_MC2_EL72xx_M_nMC_DriveData_iState:= FB_MC2_EL72xx_M_nMC_DriveData_iState +1;

	003:	// Check - MDP742 profile
			M_nMC_DriveData:= Tc3_HBI_System.cRUNNING;
			FB_MC2_EL72xx_M_nMC_DriveData_fbEcCoESdoRead(bExecute:= TRUE);
			IF FB_MC2_EL72xx_M_nMC_DriveData_fbEcCoESdoRead.bError THEN
				FB_MC2_EL72xx_M_nMC_DriveData_iState:= FB_MC2_EL72xx_M_nMC_DriveData_iState +1;
			ELSE
				IF NOT FB_MC2_EL72xx_M_nMC_DriveData_fbEcCoESdoRead.bBusy THEN
					FB_MC2_EL72xx_M_nMC_DriveData_bMDP742:= TRUE;
					FB_MC2_EL72xx_M_nMC_DriveData_bDS402:= FALSE;
					FB_MC2_EL72xx_M_nMC_DriveData_iState:= 000;
				END_IF			
			END_IF
	
	004:	// Check - DS402 profile
			M_nMC_DriveData:= Tc3_HBI_System.cRUNNING;
			FB_MC2_EL72xx_M_nMC_DriveData_fbEcCoESdoRead(bExecute:= FALSE);
			FB_MC2_EL72xx_M_nMC_DriveData_fbEcCoESdoRead(
				sNetId:= _stDriveAddress.NetID, 
				nSlaveAddr:= _stDriveAddress.SlaveAddress, 
				nSubIndex:= 16#11, 
				nIndex:= 16#2040, 
				pDstBuf:= ADR(FB_MC2_EL72xx_M_nMC_DriveData_nInt), 
				cbBufLen:= SIZEOF(FB_MC2_EL72xx_M_nMC_DriveData_nInt), 
				bExecute:= TRUE, 
				tTimeout:= T#2S);
	 
			FB_MC2_EL72xx_M_nMC_DriveData_iState:= FB_MC2_EL72xx_M_nMC_DriveData_iState +1;
			
	005:	// Check - DS402 profile
			M_nMC_DriveData:= Tc3_HBI_System.cRUNNING;
			FB_MC2_EL72xx_M_nMC_DriveData_fbEcCoESdoRead(bExecute:= TRUE);
			IF FB_MC2_EL72xx_M_nMC_DriveData_fbEcCoESdoRead.bError THEN
				M_nError(nErrorID:= FB_MC2_EL72xx_M_nMC_DriveData_fbEcCoESdoRead.nErrId);
				M_nMC_DriveData:= FB_MC2_EL72xx_M_nMC_DriveData_fbEcCoESdoRead.nErrId;
			ELSE
				IF NOT FB_MC2_EL72xx_M_nMC_DriveData_fbEcCoESdoRead.bBusy THEN
					FB_MC2_EL72xx_M_nMC_DriveData_bMDP742:= FALSE;
					FB_MC2_EL72xx_M_nMC_DriveData_bDS402:= TRUE;
					FB_MC2_EL72xx_M_nMC_DriveData_iState:= 000;
				END_IF			
			END_IF

//***********************************			
// MDP742 profile			
//***********************************			
	
	010:	// Read Internal temperatur - MDP742
			M_nMC_DriveData:= Tc3_HBI_System.cCOMPLETE;
			FB_MC2_EL72xx_M_nMC_DriveData_fbEcCoESdoRead(bExecute:= FALSE);
			FB_MC2_EL72xx_M_nMC_DriveData_fbEcCoESdoRead(
				sNetId:= _stDriveAddress.NetID, 
				nSlaveAddr:= _stDriveAddress.SlaveAddress, 
				nSubIndex:= 16#11, 
				nIndex:= 16#9010, 
				pDstBuf:= ADR(FB_MC2_EL72xx_M_nMC_DriveData_nInt), 
				cbBufLen:= SIZEOF(FB_MC2_EL72xx_M_nMC_DriveData_nInt), 
				bExecute:= TRUE, 
				tTimeout:= T#2S);
	 
			FB_MC2_EL72xx_M_nMC_DriveData_iState:= FB_MC2_EL72xx_M_nMC_DriveData_iState +1;

	011:	// Error handling - MDP742
			M_nMC_DriveData:= Tc3_HBI_System.cCOMPLETE;
			FB_MC2_EL72xx_M_nMC_DriveData_fbEcCoESdoRead(bExecute:= TRUE);
			IF FB_MC2_EL72xx_M_nMC_DriveData_fbEcCoESdoRead.bError THEN
				M_nError(nErrorID:= FB_MC2_EL72xx_M_nMC_DriveData_fbEcCoESdoRead.nErrId);
				M_nMC_DriveData:= FB_MC2_EL72xx_M_nMC_DriveData_fbEcCoESdoRead.nErrId;
			ELSE
				// Done
				IF NOT FB_MC2_EL72xx_M_nMC_DriveData_fbEcCoESdoRead.bBusy THEN
					FB_MC2_EL72xx_M_nMC_DriveData_fbEcCoESdoRead(bExecute:= FALSE);
					FB_MC2_EL72xx_M_nMC_DriveData_lrAmplifierTemperature:= UINT_TO_LREAL(FB_MC2_EL72xx_M_nMC_DriveData_nInt) / 10.0;
					FB_MC2_EL72xx_M_nMC_DriveData_iState:= FB_MC2_EL72xx_M_nMC_DriveData_iState +1;
				END_IF	
			END_IF
	
	012:	// Read Motor supply voltage - MDP742 
			M_nMC_DriveData:= Tc3_HBI_System.cCOMPLETE;
			FB_MC2_EL72xx_M_nMC_DriveData_fbEcCoESdoRead(bExecute:= FALSE);
			FB_MC2_EL72xx_M_nMC_DriveData_fbEcCoESdoRead(
				sNetId:= _stDriveAddress.NetID, 
				nSlaveAddr:= _stDriveAddress.SlaveAddress, 
				nSubIndex:= 16#12, 
				nIndex:= 16#9010, 
				pDstBuf:= ADR(FB_MC2_EL72xx_M_nMC_DriveData_nDInt), 
				cbBufLen:= SIZEOF(FB_MC2_EL72xx_M_nMC_DriveData_nDInt), 
				bExecute:= TRUE, 
				tTimeout:= T#2S);
	 
			FB_MC2_EL72xx_M_nMC_DriveData_iState:= FB_MC2_EL72xx_M_nMC_DriveData_iState +1;

	013:	// Error handling - MDP742
			M_nMC_DriveData:= Tc3_HBI_System.cCOMPLETE;
			FB_MC2_EL72xx_M_nMC_DriveData_fbEcCoESdoRead(bExecute:= TRUE);
			IF FB_MC2_EL72xx_M_nMC_DriveData_fbEcCoESdoRead.bError THEN
				M_nError(nErrorID:= FB_MC2_EL72xx_M_nMC_DriveData_fbEcCoESdoRead.nErrId);
				M_nMC_DriveData:= FB_MC2_EL72xx_M_nMC_DriveData_fbEcCoESdoRead.nErrId;
			ELSE
				// Done
				IF NOT FB_MC2_EL72xx_M_nMC_DriveData_fbEcCoESdoRead.bBusy THEN
					FB_MC2_EL72xx_M_nMC_DriveData_fbEcCoESdoRead(bExecute:= FALSE);
					FB_MC2_EL72xx_M_nMC_DriveData_lrMotorSupplyVoltage:= (DINT_TO_LREAL(FB_MC2_EL72xx_M_nMC_DriveData_nDInt)) / 1000.0;
					FB_MC2_EL72xx_M_nMC_DriveData_iState:= FB_MC2_EL72xx_M_nMC_DriveData_iState +1;
				END_IF	
			END_IF

	014:	// Read Motor temperatur - MDP742
			M_nMC_DriveData:= Tc3_HBI_System.cCOMPLETE;
			FB_MC2_EL72xx_M_nMC_DriveData_fbEcCoESdoRead(bExecute:= FALSE);
			FB_MC2_EL72xx_M_nMC_DriveData_fbEcCoESdoRead(
				sNetId:= _stDriveAddress.NetID, 
				nSlaveAddr:= _stDriveAddress.SlaveAddress, 
				nSubIndex:= 16#13, 
				nIndex:= 16#A011, 
				pDstBuf:= ADR(FB_MC2_EL72xx_M_nMC_DriveData_nDInt), 
				cbBufLen:= SIZEOF(FB_MC2_EL72xx_M_nMC_DriveData_nDInt), 
				bExecute:= TRUE, 
				tTimeout:= T#2S);
	 
			FB_MC2_EL72xx_M_nMC_DriveData_iState:= FB_MC2_EL72xx_M_nMC_DriveData_iState +1;

	015:	// Error handling - MDP742
			M_nMC_DriveData:= Tc3_HBI_System.cCOMPLETE;
			FB_MC2_EL72xx_M_nMC_DriveData_fbEcCoESdoRead(bExecute:= TRUE);
			IF FB_MC2_EL72xx_M_nMC_DriveData_fbEcCoESdoRead.bError THEN
				M_nError(nErrorID:= FB_MC2_EL72xx_M_nMC_DriveData_fbEcCoESdoRead.nErrId);
				M_nMC_DriveData:= FB_MC2_EL72xx_M_nMC_DriveData_fbEcCoESdoRead.nErrId;
			ELSE
				// Done
				IF NOT FB_MC2_EL72xx_M_nMC_DriveData_fbEcCoESdoRead.bBusy THEN
					FB_MC2_EL72xx_M_nMC_DriveData_fbEcCoESdoRead(bExecute:= FALSE);
					FB_MC2_EL72xx_M_nMC_DriveData_lrMotorTemperature:= (DINT_TO_LREAL(FB_MC2_EL72xx_M_nMC_DriveData_nDInt)) / 10.0;
					FB_MC2_EL72xx_M_nMC_DriveData_iState:= FB_MC2_EL72xx_M_nMC_DriveData_iState +1;
				END_IF	
			END_IF
	
	016:	// Done	- MDP742	
			M_nMC_DriveData:= Tc3_HBI_System.cCOMPLETE;
			FB_MC2_EL72xx_M_nMC_DriveData_iState:= 000;

//***********************************			
// DS402 profile			
//***********************************			

	020:	// Read Internal temperatur - DS402
			M_nMC_DriveData:= Tc3_HBI_System.cCOMPLETE;
			FB_MC2_EL72xx_M_nMC_DriveData_fbEcCoESdoRead(bExecute:= FALSE);
			FB_MC2_EL72xx_M_nMC_DriveData_fbEcCoESdoRead(
				sNetId:= _stDriveAddress.NetID, 
				nSlaveAddr:= _stDriveAddress.SlaveAddress, 
				nSubIndex:= 16#11, 
				nIndex:= 16#2040, 
				pDstBuf:= ADR(FB_MC2_EL72xx_M_nMC_DriveData_nInt), 
				cbBufLen:= SIZEOF(FB_MC2_EL72xx_M_nMC_DriveData_nInt), 
				bExecute:= TRUE, 
				tTimeout:= T#2S);
	 
			FB_MC2_EL72xx_M_nMC_DriveData_iState:= FB_MC2_EL72xx_M_nMC_DriveData_iState +1;

	021:	// Error handling - DS402
			M_nMC_DriveData:= Tc3_HBI_System.cCOMPLETE;
			FB_MC2_EL72xx_M_nMC_DriveData_fbEcCoESdoRead(bExecute:= TRUE);
			IF FB_MC2_EL72xx_M_nMC_DriveData_fbEcCoESdoRead.bError THEN
				M_nError(nErrorID:= FB_MC2_EL72xx_M_nMC_DriveData_fbEcCoESdoRead.nErrId);
				M_nMC_DriveData:= FB_MC2_EL72xx_M_nMC_DriveData_fbEcCoESdoRead.nErrId;
			ELSE
				// Done
				IF NOT FB_MC2_EL72xx_M_nMC_DriveData_fbEcCoESdoRead.bBusy THEN
					FB_MC2_EL72xx_M_nMC_DriveData_fbEcCoESdoRead(bExecute:= FALSE);
					FB_MC2_EL72xx_M_nMC_DriveData_lrAmplifierTemperature:= UINT_TO_LREAL(FB_MC2_EL72xx_M_nMC_DriveData_nInt) / 10.0;
					FB_MC2_EL72xx_M_nMC_DriveData_iState:= FB_MC2_EL72xx_M_nMC_DriveData_iState +1;
				END_IF	
			END_IF
	
	022:	// Read Motor supply voltage - DS402 
			M_nMC_DriveData:= Tc3_HBI_System.cCOMPLETE;
			FB_MC2_EL72xx_M_nMC_DriveData_fbEcCoESdoRead(bExecute:= FALSE);
			FB_MC2_EL72xx_M_nMC_DriveData_fbEcCoESdoRead(
				sNetId:= _stDriveAddress.NetID, 
				nSlaveAddr:= _stDriveAddress.SlaveAddress, 
				nSubIndex:= 16#12, 
				nIndex:= 16#2040, 
				pDstBuf:= ADR(FB_MC2_EL72xx_M_nMC_DriveData_nDInt), 
				cbBufLen:= SIZEOF(FB_MC2_EL72xx_M_nMC_DriveData_nDInt), 
				bExecute:= TRUE, 
				tTimeout:= T#2S);
	 
			FB_MC2_EL72xx_M_nMC_DriveData_iState:= FB_MC2_EL72xx_M_nMC_DriveData_iState +1;

	023:	// Error handling - DS402
			M_nMC_DriveData:= Tc3_HBI_System.cCOMPLETE;
			FB_MC2_EL72xx_M_nMC_DriveData_fbEcCoESdoRead(bExecute:= TRUE);
			IF FB_MC2_EL72xx_M_nMC_DriveData_fbEcCoESdoRead.bError THEN
				M_nError(nErrorID:= FB_MC2_EL72xx_M_nMC_DriveData_fbEcCoESdoRead.nErrId);
				M_nMC_DriveData:= FB_MC2_EL72xx_M_nMC_DriveData_fbEcCoESdoRead.nErrId;
			ELSE
				// Done
				IF NOT FB_MC2_EL72xx_M_nMC_DriveData_fbEcCoESdoRead.bBusy THEN
					FB_MC2_EL72xx_M_nMC_DriveData_fbEcCoESdoRead(bExecute:= FALSE);
					FB_MC2_EL72xx_M_nMC_DriveData_lrMotorSupplyVoltage:= (DINT_TO_LREAL(FB_MC2_EL72xx_M_nMC_DriveData_nDInt)) / 1000.0;
					FB_MC2_EL72xx_M_nMC_DriveData_iState:= FB_MC2_EL72xx_M_nMC_DriveData_iState +1;
				END_IF	
			END_IF

	024:	// Read Motor temperatur - DS402
			M_nMC_DriveData:= Tc3_HBI_System.cCOMPLETE;
			FB_MC2_EL72xx_M_nMC_DriveData_fbEcCoESdoRead(bExecute:= FALSE);
			FB_MC2_EL72xx_M_nMC_DriveData_fbEcCoESdoRead(
				sNetId:= _stDriveAddress.NetID, 
				nSlaveAddr:= _stDriveAddress.SlaveAddress, 
				nSubIndex:= 16#13, 
				nIndex:= 16#2031, 
				pDstBuf:= ADR(FB_MC2_EL72xx_M_nMC_DriveData_nDInt), 
				cbBufLen:= SIZEOF(FB_MC2_EL72xx_M_nMC_DriveData_nDInt), 
				bExecute:= TRUE, 
				tTimeout:= T#2S);
	 
			FB_MC2_EL72xx_M_nMC_DriveData_iState:= FB_MC2_EL72xx_M_nMC_DriveData_iState +1;

	025:	// Error handling - DS402
			M_nMC_DriveData:= Tc3_HBI_System.cCOMPLETE;
			FB_MC2_EL72xx_M_nMC_DriveData_fbEcCoESdoRead(bExecute:= TRUE);
			IF FB_MC2_EL72xx_M_nMC_DriveData_fbEcCoESdoRead.bError THEN
				M_nError(nErrorID:= FB_MC2_EL72xx_M_nMC_DriveData_fbEcCoESdoRead.nErrId);
				M_nMC_DriveData:= FB_MC2_EL72xx_M_nMC_DriveData_fbEcCoESdoRead.nErrId;
			ELSE
				// Done
				IF NOT FB_MC2_EL72xx_M_nMC_DriveData_fbEcCoESdoRead.bBusy THEN
					FB_MC2_EL72xx_M_nMC_DriveData_fbEcCoESdoRead(bExecute:= FALSE);
					FB_MC2_EL72xx_M_nMC_DriveData_lrMotorTemperature:= (DINT_TO_LREAL(FB_MC2_EL72xx_M_nMC_DriveData_nDInt)) / 10.0;
					FB_MC2_EL72xx_M_nMC_DriveData_iState:= FB_MC2_EL72xx_M_nMC_DriveData_iState +1;
				END_IF	
			END_IF
	
	026:	// Done	- DS402	
			M_nMC_DriveData:= Tc3_HBI_System.cCOMPLETE;
			FB_MC2_EL72xx_M_nMC_DriveData_iState:= 000;
	
ELSE
	FB_MC2_EL72xx_M_nMC_DriveData_iState:= 000;
END_CASE
END_METHOD

//	The result of the method is an unsigned double integer
//	0 = idle 
//	1 = coupled
//	2 = starting
//	3 = running
//	4 = aborted
// 	5 = no hardware connected
// 	6 = Spare
//	7 = pointer or index error
//	8 = mapping error
//	9 = parameter error
//	10 = complete
//	Any other number = ErrorID
METHOD PUBLIC M_nMC_Power : UDINT
VAR_INPUT
	bEnable: BOOL;
	bE_Stop: BOOL;
	bE_StopDelay: BOOL;
	bEnable_Positive: BOOL;
	bEnable_Negative: BOOL;
END_VAR
// Local variable
FB_MC2_EL72xx_M_nMC_Power_bEnable:= bEnable;
FB_MC2_EL72xx_M_nMC_Power_bE_Stop:= bE_Stop;
FB_MC2_EL72xx_M_nMC_Power_bE_StopDelay:= bE_StopDelay;
FB_MC2_EL72xx_M_nMC_Power_bEnable_Positive:= bEnable_Positive;
FB_MC2_EL72xx_M_nMC_Power_bEnable_Negative:= bEnable_Negative; 

//**********************************
// Reset 
//**********************************
IF _bReset THEN
	MEMSET(destAddr:= ADR(FB_MC2_EL72xx_M_nMC_Power_arr_nRet), fillByte:= 16#00, n:= SIZEOF(FB_MC2_EL72xx_M_nMC_Power_arr_nRet));

	// Reset all methods
	M_nMC_DriveData();
END_IF

//**********************************
// Call methodes	
//**********************************
FB_MC2_EL72xx_M_nMC_Power_fbStartDelay_TON(IN:= TRUE, PT:= T#200MS, Q=> , ET=> );
IF _stAXIS_REF.NcToPlc.AxisID > 0 OR FB_MC2_EL72xx_M_nMC_Power_fbStartDelay_TON.Q THEN
	FB_MC2_EL72xx_M_nMC_Power_arr_nRet[1]:= SUPER^.M_nMC_Power(bEnable:= FB_MC2_EL72xx_M_nMC_Power_bEnable, bE_Stop:= FB_MC2_EL72xx_M_nMC_Power_bE_Stop, bE_StopDelay:= FB_MC2_EL72xx_M_nMC_Power_bE_StopDelay, bEnable_Positive:= FB_MC2_EL72xx_M_nMC_Power_bEnable_Positive, bEnable_Negative:= FB_MC2_EL72xx_M_nMC_Power_bEnable_Negative);
	FB_MC2_EL72xx_M_nMC_Power_arr_nRet[2]:= M_nMC_DriveData();
	FB_MC2_EL72xx_M_nMC_Power_arr_nRet[3]:= M_nMC_DeadTimeComp();
ELSE
	SUPER^.M_nMC_Power(bEnable:= FALSE, bE_Stop:= FB_MC2_EL72xx_M_nMC_Power_bE_Stop, bE_StopDelay:= FB_MC2_EL72xx_M_nMC_Power_bE_StopDelay, bEnable_Positive:= FB_MC2_EL72xx_M_nMC_Power_bEnable_Positive, bEnable_Negative:= FB_MC2_EL72xx_M_nMC_Power_bEnable_Negative);
	IF FB_MC2_EL72xx_M_nMC_Power_bEnable THEN
		M_nMC_Power:= Tc3_HBI_System.cMAPPING_ERROR;		
	END_IF
	RETURN;
END_IF


//**********************************
// Error handling
//**********************************
IF _stAXIS_REF.Status.Error THEN
	M_nError(_stAXIS_REF.Status.ErrorID);
	M_nMC_Power:= _nErrorID;
ELSE
	FOR _iIdx:= 1 TO UINT_TO_INT(SIZEOF(FB_MC2_EL72xx_M_nMC_Power_arr_nRet) / SIZEOF(FB_MC2_EL72xx_M_nMC_Power_arr_nRet[1])) DO
		IF FB_MC2_EL72xx_M_nMC_Power_arr_nRet[_iIdx] > 5 AND FB_MC2_EL72xx_M_nMC_Power_arr_nRet[_iIdx] <> 10 THEN
			M_nError(nErrorID:= FB_MC2_EL72xx_M_nMC_Power_arr_nRet[_iIdx]);
			EXIT;
		END_IF
	END_FOR

	// Method return value
	IF _bError THEN
		M_nMC_Power:= _nErrorID;
	ELSE
		M_nMC_Power:= FB_MC2_EL72xx_M_nMC_Power_arr_nRet[1];
	END_IF

END_IF
END_METHOD

PROPERTY PUBLIC P_rAmplifierTemperature : REAL
GET
P_rAmplifierTemperature:= LREAL_TO_REAL(FB_MC2_EL72xx_M_nMC_DriveData_lrAmplifierTemperature);
END_GET
END_PROPERTY

PROPERTY PUBLIC P_rMotorSupplyVoltage : REAL
GET
P_rMotorSupplyVoltage:= LREAL_TO_REAL(FB_MC2_EL72xx_M_nMC_DriveData_lrMotorSupplyVoltage);
END_GET
END_PROPERTY

PROPERTY PUBLIC P_rMotorTemperature : REAL
GET
P_rMotorTemperature:= LREAL_TO_REAL(FB_MC2_EL72xx_M_nMC_DriveData_lrMotorTemperature);
END_GET
END_PROPERTY

END_FUNCTION_BLOCK

// MOTION/POUs/FBs/Compact/FB_MC2_Compact_AX8000
//------------------------------------------------------------------------------------------
//                                                                                        	
//***************************** Beckhoff TwinCAT Examples **********************************
//                                                                                        	
//************************************* WARNING ********************************************
// This program is only an example. If it is used as a control program in any real        	
// application, Beckhoff is not responsible for any malfunction, loss or damage           	
// which could arise by using this program!                                               	
//                                                                                        	
//*************************************  Program Info. *************************************
//                                                                                        	
// PLC program name:    	FB_MC2_Compact_AX8000 (FB)               	                           	
// Hardware platform:      	TwinCat PTP v3.1 4022				                          	                                 	
//                                                                                        	
// ======================================================================================== 
//         Version       Date                        Remarks                              	
// ======================================================================================== 
//         3.1           27 feb 2018                 First release of this example        	
//
// ======================================================================================== 
//                                                                                        	
//******************************* Aims OF this PLC PROGRAM *********************************
//                                                                                        	
// MC2 AX8000 servo axis 						 			                               	
//                                                                                        	
//----------------------------------------------------------------------------------------- 
FUNCTION_BLOCK FB_MC2_Compact_AX8000 EXTENDS FB_MC2_Compact 
VAR
	FB_MC2_Compact_AX8000_M_nMC_DriveData_iState: INT;	
	FB_MC2_Compact_AX8000_M_nMC_DriveData_lrActualMainVoltage: LREAL;
	FB_MC2_Compact_AX8000_M_nMC_DriveData_lrAmplifierTemperature: LREAL;
	FB_MC2_Compact_AX8000_M_nMC_DriveData_lrMotorTemperature: LREAL;
	FB_MC2_Compact_AX8000_M_nMC_DriveData_fbCoERead: Tc2_MC2_Drive.FB_CoERead;
	FB_MC2_Compact_AX8000_M_nMC_DriveData_fbCoEWrite: Tc2_MC2_Drive.FB_CoEWrite;
	FB_MC2_Compact_AX8000_M_nMC_DriveData_iValue: INT;
	FB_MC2_Compact_AX8000_M_nMC_DriveData_rValue: REAL;

	FB_MC2_Compact_AX8000_M_nMC_Power_bEnable: BOOL;
	FB_MC2_Compact_AX8000_M_nMC_Power_bE_Stop: BOOL;
	FB_MC2_Compact_AX8000_M_nMC_Power_bE_StopDelay: BOOL;
	FB_MC2_Compact_AX8000_M_nMC_Power_bEnable_Positive: BOOL;
	FB_MC2_Compact_AX8000_M_nMC_Power_bEnable_Negative: BOOL;
	FB_MC2_Compact_AX8000_M_nMC_Power_fbStartDelay_TON: Tc2_Standard.TON;
	FB_MC2_Compact_AX8000_M_nMC_Power_arr_nRet: ARRAY[1..4] OF UDINT;
	
	FB_MC2_Compact_AX8000_M_nReset_iState: INT;
	FB_MC2_Compact_AX8000_M_nReset_fbExecute_R_TRIG: Tc2_Standard.R_TRIG;
	FB_MC2_Compact_AX8000_M_nReset_nStatus: UDINT;
END_VAR

//	The result of the method is an unsigned double integer
//	0 = idle 
//	1 = coupled
//	2 = starting
//	3 = running
//	4 = aborted
// 	5 = no hardware connected
// 	6 = Spare
//	7 = pointer or index error
//	8 = mapping error
//	9 = parameter error
//	10 = complete
//	Any other number = ErrorID
METHOD PRIVATE M_nMC_DriveData : UDINT
//**********************************
// Reset 
//**********************************
IF _bReset THEN
	IF _bError THEN
		FB_MC2_Compact_AX8000_M_nMC_DriveData_fbCoERead(Execute:= FALSE, Axis:= _stAXIS_REF); 
		FB_MC2_Compact_AX8000_M_nMC_DriveData_fbCoEWrite(Execute:= FALSE, Axis:= _stAXIS_REF);
	END_IF
	RETURN;
END_IF

// No hardware connected
IF NOT _bHardwareConnected THEN
	FB_MC2_Compact_AX8000_M_nMC_DriveData_lrActualMainVoltage:= 0.0;				// Drive Main voltage
	FB_MC2_Compact_AX8000_M_nMC_DriveData_lrAmplifierTemperature:= 0.0;				// Drive temperatur
	FB_MC2_Compact_AX8000_M_nMC_DriveData_lrMotorTemperature:= 0.0;					// Motor temperatur
	FB_MC2_Compact_AX8000_M_nMC_DriveData_fbCoERead(Execute:= FALSE, Axis:= _stAXIS_REF); 
	FB_MC2_Compact_AX8000_M_nMC_DriveData_fbCoEWrite(Execute:= FALSE, Axis:= _stAXIS_REF);
	FB_MC2_Compact_AX8000_M_nMC_DriveData_iState:= 000;
	M_nMC_DriveData:= Tc3_HBI_System.cNO_HARDWARE_CONNECTED;
	RETURN;
END_IF


//**********************************
// Main sequence
//**********************************

CASE FB_MC2_Compact_AX8000_M_nMC_DriveData_iState OF
	
	000:	// Init
			FB_MC2_Compact_AX8000_M_nMC_DriveData_fbCoERead(Execute:= FALSE, Axis:= _stAXIS_REF); 
			FB_MC2_Compact_AX8000_M_nMC_DriveData_fbCoEWrite(Execute:= FALSE, Axis:= _stAXIS_REF);
			FB_MC2_Compact_AX8000_M_nMC_DriveData_iValue:= 0;
			FB_MC2_Compact_AX8000_M_nMC_DriveData_rValue:= 0.0;
			M_nMC_DriveData:= Tc3_HBI_System.cSTARTING;

			// Simulations axis 
			IF _stAXIS_REF.NcToPlc.AxisID > 0 THEN
				IF _stAXIS_REF.Status.OpMode.SimulationAxis THEN
					FB_MC2_Compact_AX8000_M_nMC_DriveData_lrActualMainVoltage:= 0.0;			// Drive Main voltage
					FB_MC2_Compact_AX8000_M_nMC_DriveData_lrAmplifierTemperature:= 0.0;			// Drive temperatur
					FB_MC2_Compact_AX8000_M_nMC_DriveData_lrMotorTemperature:= 0.0;				// Motor temperatur
					M_nMC_DriveData:= Tc3_HBI_System.cNO_HARDWARE_CONNECTED;
				ELSE
					// Axis connected to Hardware
					IF _bHardwareConnected THEN
						M_nMC_DriveData:= Tc3_HBI_System.cCOMPLETE;
						FB_MC2_Compact_AX8000_M_nMC_DriveData_iState:= FB_MC2_Compact_AX8000_M_nMC_DriveData_iState +1;
					ELSE
						FB_MC2_Compact_AX8000_M_nMC_DriveData_lrActualMainVoltage:= 0.0;		// Drive Main voltage
						FB_MC2_Compact_AX8000_M_nMC_DriveData_lrAmplifierTemperature:= 0.0;		// Drive temperatur
						FB_MC2_Compact_AX8000_M_nMC_DriveData_lrMotorTemperature:= 0.0;			// Motor temperatur
						M_nMC_DriveData:= Tc3_HBI_System.cNO_HARDWARE_CONNECTED;
					END_IF
				END_IF
			ELSE
				FB_MC2_Compact_AX8000_M_nMC_DriveData_lrActualMainVoltage:= 0.0;				// Drive Main voltage
				FB_MC2_Compact_AX8000_M_nMC_DriveData_lrAmplifierTemperature:= 0.0;				// Drive temperatur
				FB_MC2_Compact_AX8000_M_nMC_DriveData_lrMotorTemperature:= 0.0;					// Motor temperatur
				M_nMC_DriveData:= Tc3_HBI_System.cNO_HARDWARE_CONNECTED;
			END_IF
	
//**************************************************************************
// Init values
//**************************************************************************

	001:	// Set motor temp type - 0x32C0:0F
			M_nMC_DriveData:= Tc3_HBI_System.cRUNNING;
			FB_MC2_Compact_AX8000_M_nMC_DriveData_iValue:= 1;
			FB_MC2_Compact_AX8000_M_nMC_DriveData_fbCoEWrite(
				NetId:= '', 
				Index:= 16#32C0 + (16#0400 * _stDriveAddress.Channel), 
				SubIndex:= 16#0F, 
				pSrcBuf:= ADR(FB_MC2_Compact_AX8000_M_nMC_DriveData_iValue), 
				BufLen:= SIZEOF(FB_MC2_Compact_AX8000_M_nMC_DriveData_iValue), 
				Execute:= TRUE, 
				Timeout:= , 
				CompleteAccess:= , 
				Axis:= _stAXIS_REF, 
				Busy=> , 
				Error=> , 
				AdsErrId=> , 
				CANopenErrId=> );	

			// Error handling
			IF FB_MC2_Compact_AX8000_M_nMC_DriveData_fbCoEWrite.Error THEN
				M_nError(FB_MC2_Compact_AX8000_M_nMC_DriveData_fbCoEWrite.AdsErrId);
				M_nMC_DriveData:= FB_MC2_Compact_AX8000_M_nMC_DriveData_fbCoEWrite.AdsErrId;
			ELSE
				// Done
				IF NOT FB_MC2_Compact_AX8000_M_nMC_DriveData_fbCoEWrite.Busy THEN
					FB_MC2_Compact_AX8000_M_nMC_DriveData_fbCoEWrite(Execute:= FALSE, Axis:= _stAXIS_REF);
					FB_MC2_Compact_AX8000_M_nMC_DriveData_iValue:= 0;
					FB_MC2_Compact_AX8000_M_nMC_DriveData_iState:= 010;
				END_IF
			END_IF
			
//**************************************************************************
// Running values
//**************************************************************************

	010:	// Read motor temp - 0x32C1:06			
			M_nMC_DriveData:= Tc3_HBI_System.cCOMPLETE;
			FB_MC2_Compact_AX8000_M_nMC_DriveData_fbCoERead(
				NetId:= '', 
				Index:= 16#32C1 + (16#0400 * _stDriveAddress.Channel), 
				SubIndex:= 16#06, 
				pDstBuf:= ADR(FB_MC2_Compact_AX8000_M_nMC_DriveData_rValue), 
				BufLen:= SIZEOF(FB_MC2_Compact_AX8000_M_nMC_DriveData_rValue), 
				Execute:= TRUE, 
				Timeout:= , 
				CompleteAccess:= , 
				Axis:= _stAXIS_REF, 
				Busy=> , 
				Error=> , 
				AdsErrId=> , 
				CANopenErrId=> );
		
			// Error handling
			IF FB_MC2_Compact_AX8000_M_nMC_DriveData_fbCoERead.Error THEN
				M_nError(FB_MC2_Compact_AX8000_M_nMC_DriveData_fbCoERead.AdsErrId);
				M_nMC_DriveData:= FB_MC2_Compact_AX8000_M_nMC_DriveData_fbCoERead.AdsErrId;
			ELSE
				// Done
				IF NOT FB_MC2_Compact_AX8000_M_nMC_DriveData_fbCoERead.Busy THEN
					FB_MC2_Compact_AX8000_M_nMC_DriveData_lrMotorTemperature:= REAL_TO_LREAL(FB_MC2_Compact_AX8000_M_nMC_DriveData_rValue);
					FB_MC2_Compact_AX8000_M_nMC_DriveData_fbCoERead(Execute:= FALSE, Axis:= _stAXIS_REF);
					FB_MC2_Compact_AX8000_M_nMC_DriveData_rValue:= 0.0;
					FB_MC2_Compact_AX8000_M_nMC_DriveData_iState:= FB_MC2_Compact_AX8000_M_nMC_DriveData_iState +1;
				END_IF
			END_IF

	011:	// Read IGBT temp - 0x3001:02			
			M_nMC_DriveData:= Tc3_HBI_System.cCOMPLETE;
			FB_MC2_Compact_AX8000_M_nMC_DriveData_fbCoERead(
				NetId:= '', 
				Index:= 16#3001 + (16#0400 * _stDriveAddress.Channel), 
				SubIndex:= 16#02, 
				pDstBuf:= ADR(FB_MC2_Compact_AX8000_M_nMC_DriveData_iValue), 
				BufLen:= SIZEOF(FB_MC2_Compact_AX8000_M_nMC_DriveData_iValue), 
				Execute:= TRUE, 
				Timeout:= , 
				CompleteAccess:= , 
				Axis:= _stAXIS_REF, 
				Busy=> , 
				Error=> , 
				AdsErrId=> , 
				CANopenErrId=> );
		
			// Error handling
			IF FB_MC2_Compact_AX8000_M_nMC_DriveData_fbCoERead.Error THEN
				M_nError(FB_MC2_Compact_AX8000_M_nMC_DriveData_fbCoERead.AdsErrId);
				M_nMC_DriveData:= FB_MC2_Compact_AX8000_M_nMC_DriveData_fbCoERead.AdsErrId;
			ELSE
				// Done
				IF NOT FB_MC2_Compact_AX8000_M_nMC_DriveData_fbCoERead.Busy THEN
					FB_MC2_Compact_AX8000_M_nMC_DriveData_lrAmplifierTemperature:= INT_TO_LREAL(FB_MC2_Compact_AX8000_M_nMC_DriveData_iValue);
					FB_MC2_Compact_AX8000_M_nMC_DriveData_fbCoERead(Execute:= FALSE, Axis:= _stAXIS_REF);
					FB_MC2_Compact_AX8000_M_nMC_DriveData_iValue:= 0;
					FB_MC2_Compact_AX8000_M_nMC_DriveData_iState:= FB_MC2_Compact_AX8000_M_nMC_DriveData_iState +1;
				END_IF
			END_IF

			
	012:	//
			FB_MC2_Compact_AX8000_M_nMC_DriveData_iState:= 010;
	
			
ELSE
	FB_MC2_Compact_AX8000_M_nMC_DriveData_iState:= 000;
END_CASE
END_METHOD

//	The result of the method is an unsigned double integer
//	0 = idle 
//	1 = coupled
//	2 = starting
//	3 = running
//	4 = aborted
// 	5 = no hardware connected
// 	6 = Spare
//	7 = pointer or index error
//	8 = mapping error
//	9 = parameter error
//	10 = complete
//	Any other number = ErrorID
METHOD PUBLIC M_nMC_Power : UDINT
VAR_INPUT
	bEnable: BOOL;
	bE_Stop: BOOL;
	bE_StopDelay: BOOL;
	bEnable_Positive: BOOL;
	bEnable_Negative: BOOL;
END_VAR
// Local variable
FB_MC2_Compact_AX8000_M_nMC_Power_bEnable:= bEnable;
FB_MC2_Compact_AX8000_M_nMC_Power_bE_Stop:= bE_Stop;
FB_MC2_Compact_AX8000_M_nMC_Power_bE_StopDelay:= bE_StopDelay; 
FB_MC2_Compact_AX8000_M_nMC_Power_bEnable_Positive:= bEnable_Positive;
FB_MC2_Compact_AX8000_M_nMC_Power_bEnable_Negative:= bEnable_Negative;

//**********************************
// Reset 
//**********************************
IF _bReset THEN
	MEMSET(destAddr:= ADR(FB_MC2_Compact_AX8000_M_nMC_Power_arr_nRet), fillByte:= 16#00, n:= SIZEOF(FB_MC2_Compact_AX8000_M_nMC_Power_arr_nRet));

	M_nMC_DriveData();
END_IF

//**********************************
// Call methods 
//**********************************
FB_MC2_Compact_AX8000_M_nMC_Power_fbStartDelay_TON(IN:= TRUE, PT:= T#200MS, Q=> , ET=> );
IF FB_MC2_Compact_AX8000_M_nMC_Power_fbStartDelay_TON.Q THEN
	IF _stAXIS_REF.NcToPlc.AxisID > 0 THEN
		FB_MC2_Compact_AX8000_M_nMC_Power_arr_nRet[1]:= SUPER^.M_nMC_Power(bEnable:= FB_MC2_Compact_AX8000_M_nMC_Power_bEnable, bE_Stop:= FB_MC2_Compact_AX8000_M_nMC_Power_bE_Stop, bE_StopDelay:= FB_MC2_Compact_AX8000_M_nMC_Power_bE_StopDelay, bEnable_Positive:= FB_MC2_Compact_AX8000_M_nMC_Power_bEnable_Positive, bEnable_Negative:= FB_MC2_Compact_AX8000_M_nMC_Power_bEnable_Negative);
		FB_MC2_Compact_AX8000_M_nMC_Power_arr_nRet[2]:= M_nMC_DriveData();				
	ELSE
		SUPER^.M_nMC_Power(bEnable:= FALSE, bE_Stop:= FB_MC2_Compact_AX8000_M_nMC_Power_bE_Stop, bE_StopDelay:= FB_MC2_Compact_AX8000_M_nMC_Power_bE_StopDelay, bEnable_Positive:= FB_MC2_Compact_AX8000_M_nMC_Power_bEnable_Positive, bEnable_Negative:= FB_MC2_Compact_AX8000_M_nMC_Power_bEnable_Negative);
		IF FB_MC2_Compact_AX8000_M_nMC_Power_bEnable THEN
			M_nMC_Power:= Tc3_HBI_System.cMAPPING_ERROR;
		END_IF
		RETURN;
	END_IF
END_IF


//**********************************
// Error handling
//**********************************
IF _stAXIS_REF.Status.Error THEN
	M_nError(_stAXIS_REF.Status.ErrorID);
	M_nMC_Power:= _nErrorID;
ELSE
	FOR _iIdx:= 1 TO UINT_TO_INT(SIZEOF(FB_MC2_Compact_AX8000_M_nMC_Power_arr_nRet) / SIZEOF(FB_MC2_Compact_AX8000_M_nMC_Power_arr_nRet[1])) DO
		IF FB_MC2_Compact_AX8000_M_nMC_Power_arr_nRet[_iIdx] > 5 AND FB_MC2_Compact_AX8000_M_nMC_Power_arr_nRet[_iIdx] <> 10 THEN
			M_nError(nErrorID:= FB_MC2_Compact_AX8000_M_nMC_Power_arr_nRet[_iIdx]);
			EXIT;
		END_IF
	END_FOR

	// Method return value
	IF _bError THEN
		M_nMC_Power:= _nErrorID;
	ELSE
		M_nMC_Power:= FB_MC2_Compact_AX8000_M_nMC_Power_arr_nRet[1];
	END_IF

END_IF
END_METHOD

//	The result of the method is an unsigned double integer
//	0 = idle 
//	1 = coupled
//	2 = starting
//	3 = running
//	4 = aborted
// 	5 = no hardware connected
// 	6 = Spare
//	7 = pointer or index error
//	8 = mapping error
//	9 = parameter error
//	10 = complete
//	Any other number = ErrorID
METHOD PUBLIC M_nReset : UDINT
VAR_INPUT
	bExecute: BOOL;
END_VAR
//**********************************
// Wait for execute
//**********************************
FB_MC2_Compact_AX8000_M_nReset_fbExecute_R_TRIG(CLK:= bExecute);
IF FB_MC2_Compact_AX8000_M_nReset_fbExecute_R_TRIG.Q THEN
	SUPER^.M_nReset(bExecute:= FALSE);
	FB_MC2_Compact_AX8000_M_nReset_iState:= 001;
END_IF


//**********************************
// Main sequence
//**********************************
CASE FB_MC2_Compact_AX8000_M_nReset_iState OF

	000: 	// Do nothing

	001:	// Reset father	
			M_nReset:= Tc3_HBI_System.cRUNNING;
			FB_MC2_Compact_AX8000_M_nReset_nStatus:= SUPER^.M_nReset(bExecute:= TRUE); 
			IF FB_MC2_Compact_AX8000_M_nReset_nStatus = Tc3_HBI_System.cCOUPLED OR FB_MC2_Compact_AX8000_M_nReset_nStatus = Tc3_HBI_System.cCOMPLETE THEN		
				SUPER^.M_nReset(bExecute:= FALSE);
				IF _stAXIS_REF.Status.Coupled THEN
					FB_MC2_Compact_AX8000_M_nReset_iState:= 020;
				ELSE
					FB_MC2_Compact_AX8000_M_nReset_iState:= 030;
				END_IF
			END_IF

	020:	// Coupled
			M_nReset:= Tc3_HBI_System.cCOUPLED;
			IF NOT bExecute THEN
				SUPER^.M_nReset(bExecute:= FALSE);
				FB_MC2_Compact_AX8000_M_nReset_iState:= 000;
			END_IF	

	030: 	// Done
			M_nReset:= Tc3_HBI_System.cCOMPLETE;
			IF NOT bExecute THEN
				SUPER^.M_nReset(bExecute:= FALSE);
				FB_MC2_Compact_AX8000_M_nReset_iState:= 000;
			END_IF	
		
ELSE
	FB_MC2_Compact_AX8000_M_nReset_iState:= 000;
END_CASE
END_METHOD

PROPERTY PUBLIC P_rActualMainVoltage : REAL
GET
P_rActualMainVoltage:= LREAL_TO_REAL(FB_MC2_Compact_AX8000_M_nMC_DriveData_lrActualMainVoltage);
END_GET
END_PROPERTY

PROPERTY PUBLIC P_rAmplifierTemperature : REAL
GET
P_rAmplifierTemperature:= LREAL_TO_REAL(FB_MC2_Compact_AX8000_M_nMC_DriveData_lrAmplifierTemperature);
END_GET
END_PROPERTY

PROPERTY PUBLIC P_rMotorTemperature : REAL
GET
P_rMotorTemperature:= LREAL_TO_REAL(FB_MC2_Compact_AX8000_M_nMC_DriveData_lrMotorTemperature);
END_GET
END_PROPERTY

END_FUNCTION_BLOCK
